# B&R Automation Studio project TD52 (part 99)

### module_GC.typ
```iecst
TYPE
	MM2VIS_Struct : 	STRUCT
		tCtrGenPF_Out : _tGeACtrOut; (* Controller to visulization out structure *) (*OldName:new pv;Cycle:5*)
		tCtr_Q_Out : _tGeACtrOut; (* Controller to visulization out structure *) (*OldName:new pv;Cycle:5*)
		bP_CosPCtr_Red_F_Hi : BOOL; (* power reduction by generator frequency high active *) (*OldName:bPowRedGenFrqH;Cycle:5*)
		bP_CosPCtr_Red_F_Lo : BOOL; (* power reduction by generator frequency low active *) (*OldName:bPowRedGenFrqL;Cycle:5*)
		bP_CosPCtr_Red_U_Hi : BOOL; (* power reduction by generator voltage high active *) (*OldName:bPowRedGenSpgH;Cycle:5*)
		bP_CosPCtr_Red_U_Lo : BOOL; (* power reduction by generator voltage low active *) (*OldName:bPowRedGenSpgL;Cycle:5*)
		bPF_Ctrl_Ena : BOOL; (* plant controller No. 13 enabled *) (*OldName:bPlantCtr13;Cycle:5*)
		rAng_CosPCtr_LimCalc : REAL; (* calculated limit polar wheel angle for power factor controller *) (*OldName:rQgLimit;Cycle:5*)
		rAng_CosPCtr_LimCalcVis : REAL; (*  Q- limit for visualization  *) (*OldName:ssQLimVis;Cycle:5*)
		rAng_CosPCtr_MinCalc : REAL; (* calculated minimum polar wheel angle for trip (LOSS OF EXCITATION) *) (*OldName:rQgErregerausfall;Cycle:5*)
		rAng_CosPCtr_MinCalcVis : REAL; (*  Q- trip limit for visualization  *) (*OldName:ssQTripVis;Cycle:5*)
		rP_Red_CosPCtr_F : REAL; (* power reduction by generator frequency *) (*OldName:ssPowerRedGenFrq;Cycle:5*)
		rP_Red_CosPCtr_T : REAL; (* power reduction by generator winding temperature *) (*OldName:ssPowerRedGenTemp;Cycle:5*)
		rP_Red_CosPCtr_U : REAL; (* power reduction by generator voltage *) (*OldName:ssPowerRedGenSpg;Cycle:5*)
		rP_Gen_ppt : REAL; (* nominal power in parts per thousand *) (*OldName:PN_PROM;Cycle:5*)
		rPF_CosPCtr_LimCalc1 : REAL; (* calculated reactive power trip limit of power 0 (zero) *) (*OldName:rQgTrip0;Cycle:5*)
		rPF_CosPCtr_LimCalc2 : REAL; (* calculated reactive power trip limit of nominal power 0 (PN_GASART) *) (*OldName:rQgTripN;Cycle:5*)
		rPF_CosPCtr_MinCalc1 : REAL; (* calculated reactive power limit of power 0 (zero) *) (*OldName:rQgLimit0;Cycle:5*)
		rPF_CosPCtr_MinCalc2 : REAL; (* calculated reactive power limit of nominal power 0 (PN_GASART) *) (*OldName:rQgLimitN;Cycle:5*)
		rPF_CosPCtr_Set_Ctr13 : REAL; (* set point value for plant controller *) (*OldName:ssContr_PF_SOLL;Cycle:5*)
		rPF_CosPCtr_Set_Vis : REAL; (* enable power factor input in visualization (picture 88) *) (*OldName:usPF_input_vis;Cycle:5*)
		rPF_CosPCtr_VisLine1 : REAL; (* value for visualization *) (*OldName:ucVisLine1_P14;Cycle:5*)
		rPF_GenCtr_Act : REAL; (* power factor generator controller actual value  *) (*OldName:ssContr_IST;Cycle:5*)
		rPF_GenCtr_Set : REAL; (* power factor generator controller set point  *) (*OldName:ssContr_SOLL;Cycle:5*)
		rQ_CosPCtr_Set : REAL; (* set point of reactive power for PF- controller on XT *) (*OldName:ssQSoll;Cycle:5*)
		rT_Gen_Bear_A_Act : REAL; (*Temperature generator bearing A*) (*OldName:ANA.LAG1;Cycle:5*)
		rT_Gen_Bear_B_Act : REAL; (*Temperature generator bearing B*) (*OldName:ANA.LAG2;Cycle:5*)
		rT_Gen_Wind_Act_L1 : REAL; (* generator winding temperature signal, winding phase 1 *) (*OldName:ANA.WICK1;Cycle:5*)
		rT_Gen_Wind_Act_L2 : REAL; (* generator winding temperature signal, winding phase 2 *) (*OldName:ANA.WICK2;Cycle:5*)
		rT_Gen_Wind_Act : REAL; (*generator winding temperature signal*) (*OldName:ANA.WICK;Cycle:;*)
		rU_Gen_Exc : REAL; (*Generator excitation voltage*) (*OldName:ANA.ERREG;Cycle:5;*)
		rT_Gen_Wind_Act_L3 : REAL; (* generator winding temperature signal, winding phase 3 *) (*OldName:ANA.WICK3;Cycle:5*)
		bOilSkid_Fan_Dem : BOOL; (*OilSkid - demand of fan (TRUE = on)*) (*OldName:newPv; Cycle:5;*)
		bOilSkid_Heater_Dem : BOOL; (*OilSkid - demand of heater (TRUE = on)*) (*OldName:newPv; Cycle:5;*)
		bOilSkid_PumpC_Dem : BOOL; (*OilSkid - demand of circulation pump (TRUE = on)*) (*OldName:newPv; Cycle:5;*)
		bOilSkid_PumpLP_Dem : BOOL; (*OilSkid - demand of low pressure pump (TRUE = on)*) (*OldName:newPv; Cycle:5;*)
		bOilSkid_PumpHP_Dem : BOOL; (*OilSkid - demand of high pressure pump (TRUE = on)*) (*OldName:newPv; Cycle:5;*)
		rPr_OilSkid_HP_DE : REAL; (*OilSkid - oil pressure in high pressure circuit to DE bearing [bar]*) (*OldName:newPv; Cycle:5;*)
		rPr_OilSkid_HP_NDE : REAL; (*OilSkid - oil pressure in high pressure circuit to NDE bearing [bar]*) (*OldName:newPv; Cycle:5;*)
		rT_OilSkid_Tank : REAL; (*OilSkid - tank temperature [°C]*) (*OldName:newPv; Cycle:5;*)
		rT_OilSkid_Supply : REAL; (*OilSkid - supply temperature [°C]*) (*OldName:newPv; Cycle:5;*)
		rLev_OilSkid_Tank : REAL; (*OilSkid - tank level [%]*) (*OldName:newPv; Cycle:5;*)
		rFlow_OilSkid_DE : REAL; (*OilSkid - oil flow to DE bearing [l/min]*) (*OldName:newPv; Cycle:5;*)
		rFlow_OilSkid_NDE : REAL; (*OilSkid - oil flow to NDE bearing [l/min]*) (*OldName:newPv; Cycle:5;*)
		rF_GenBear_DE1 : REAL; (*AI vibration generator bearing drive end 1*) (*Oldname:newPv;Cycle:5;*)
		rF_GenBear_DE2 : REAL; (*AI vibration generator bearing drive end 2*) (*Oldname:newPv;Cycle:5;*)
		rF_GenBear_NDE1 : REAL; (*AI vibration generator bearing non drive end 1*) (*Oldname:newPv;Cycle:5;*)
		rF_GenBear_NDE2 : REAL; (*AI vibration generator bearing non drive end 2*) (*Oldname:newPv;Cycle:5;*)
		rGen_T_In : REAL; (*AI generator air inlet temperature*) (*Oldname:t_GenAirIn;Cycle:5;*)
		rGen_T_In2 : REAL; (*AI generator air inlet temperature 2*) (*Oldname:newPv;Cycle:5;*)
		rT_GenAirOut : REAL; (*AI generator air outlet temperature*) (*Oldname:t_GenAirOut;Cycle:5;*)
		rQ_AVR_Set_Norm : REAL; (*reactive power setpoint [%]*) (*Oldname:newPv;Cycle:5;*)
		bSel_AVR_Set : BOOL; (*Q controller enabled*) (*Oldname:newPv;Cycle:5;*)
		bQ_Lim_On : BOOL; (*Q_Set is limited, Q_Limiter is working*) (*Oldname:newPv;Cycle:5;*)
		rQS_POC : REAL; (*Q/Sn diagram Y(graph)-value for point of control(POC)*) (*Oldname:newPv;Cycle:5;*)
		rPF_POC_Act_lin : REAL; (*PF diagram Y(graph)-value for point of control(POC)*) (*Oldname:newPv;Cycle:5;*)
		bU_Gen_Inc : BOOL; (* DI voltage adjustment external (increasing)*)
		bU_Gen_Dec : BOOL; (* DI voltage adjustment external (decreasing)*)
		bMsg1036 : BOOL; (*Generator over load/short circuit, Trip *) (*OldName:M_ULKS;Cycle:5*)
		bMsg1037 : BOOL; (*Generator winding temperature maximum, Trip *) (*OldName:AN_GWTA;Cycle:5*)
		bMsg1038 : BOOL; (*Generator reverse power, Trip *) (*OldName:M_RLSG;Cycle:5*)
		bMsg1062 : BOOL; (*measuring signal failure excitation voltage *) (*OldName:MS_EREG;Cycle:5*)
		bMsg1073 : BOOL; (*MMD: overload/short circuit *) (*OldName:ALM[1073];Cycle:5*)
		bMsg1109 : BOOL; (*loss of excitation (trip) *) (*OldName:bErregerAusfall;Cycle:5*)
		bMsg1110 : BOOL; (*Generator frequency low, Trip *) (*OldName:M_GFZN;Cycle:5*)
		bMsg1111 : BOOL; (*Generator frequency high, Trip *) (*OldName:M_GFZH;Cycle:5*)
		bMsg1112 : BOOL; (*Neutral current high, Trip *) (*OldName:M_INULL;Cycle:5*)
		bMsg1113 : BOOL; (*Generator power measuring signal failure*) (*OldName:M_PIST;Cycle:5*)
		bMsg1121 : BOOL; (* generator winding temperature maximum phase 1, Trip *) (*OldName:AN_GWA1;Cycle:5*)
		bMsg1122 : BOOL; (* generator winding temperature maximum phase 2, Trip *) (*OldName:AN_GWA2;Cycle:5*)
		bMsg1123 : BOOL; (* generator winding temperature maximum phase 3, Trip *) (*OldName:AN_GWA3;Cycle:5*)
		bMsg1124 : BOOL; (* generator bearing temperature maximum bearing A, Trip *) (*OldName:AN_LAGA1;Cycle:5*)
		bMsg1125 : BOOL; (* generator bearing temperature maximum bearing B, Trip *) (*OldName:AN_LAGA2;Cycle:5*)
		bMsg1126 : BOOL; (* generator voltage low, Trip *) (*OldName:M_GUZN;Cycle:5*)
		bMsg1127 : BOOL; (* generator voltage high, Trip *) (*OldName:M_GUZH;Cycle:5*)
		bMsg1132 : BOOL; (*Differential protection, Trip*) (*OldName:M_Diff;Cycle:5*)
		bMsg1134 : BOOL; (* Earth failure, Trip *) (*OldName:M_ERDS;Cycle:5*)
		bMsg1143 : BOOL; (* Voltage negative sequence (Voltage asymmetry), Trip *) (*OldName:M_UASY;Cycle:5*)
		bMsg1144 : BOOL; (* Current negative sequnece (Current asymmetrt), Trip *) (*OldName:M_IASY;Cycle:5*)
		bMsg1154 : BOOL; (* generator winding temperature maximum phase 1, Warning *) (*OldName:AN_GWW1;Cycle:5*)
		bMsg1155 : BOOL; (* generator winding temperature maximum phase 2, Warning *) (*OldName:AN_GWW2;Cycle:5*)
		bMsg1156 : BOOL; (* generator winding temperature maximum phase 3, Warning *) (*OldName:AN_GWW3;Cycle:5*)
		bMsg1157 : BOOL; (* generator bearing temperature maximum bearing A, Warning *) (*OldName:AN_LAGW1;Cycle:5*)
		bMsg1158 : BOOL; (* generator bearing temperature maximum bearing B, Warning *) (*OldName:AN_LAGW2;Cycle:5*)
		bMsg1185 : BOOL; (* generator winding temperature maximum, Warning *) (*OldName:AN_GWTW;Cycle:5*)
		bMsg2100 : BOOL; (* Differential protection, Warning *) (*OldName:M_STDIFF;Cycle:5*)
		bMsg2105 : BOOL; (* measuring signal failure winding temperature *) (*OldName:MS_GWT;Cycle:5*)
		bMsg2106 : BOOL; (* measuring signal failure winding temperature phase 1 *) (*OldName:MS_GWT1;Cycle:5*)
		bMsg2107 : BOOL; (* measuring signal failure winding temperature phase 2 *) (*OldName:MS_GWT2;Cycle:5*)
		bMsg2108 : BOOL; (* measuring signal failure winding temperature phase 3 *) (*OldName:MS_GWT3;Cycle:5*)
		bMsg2109 : BOOL; (* measuring signal failure bearing temperature bearing A *) (*OldName:MS_LAG1;Cycle:5*)
		bMsg2110 : BOOL; (* measuring signal failure bearing temperature bearing B *) (*OldName:MS_LAG2;Cycle:5*)
		bMsg2115 : BOOL; (* Generator voltage regulator failure *) (*OldName:Not-found;Cycle:5*)
		bMsg2156 : BOOL; (* B2156 Q-RED by winding temperature limit *) (*OldName:RPSDIA[35];Cycle:5*)
		bMsg2157 : BOOL; (* B2157 Q-limit by polar wheel angle *) (*OldName:RPSDIA[36];Cycle:5*)
		bMsg2202 : BOOL; (*generator DE bearing displacement*) (*OldName:newPv;Cycle:5*)
		bMsg2203 : BOOL; (*generator NDE bearing displacement*) (*OldName:newPv;Cycle:5*)
		bMsg2204 : BOOL; (*measuring signal failure displacement sensor 1 generator DE bearing*) (*OldName:newPv;Cycle:5*)
		bMsg2205 : BOOL; (*measuring signal failure displacement sensor 2 generator DE bearing*) (*OldName:newPv;Cycle:5*)
		bMsg2206 : BOOL; (*measuring signal failure displacement sensor 1 generator NDE bearing*) (*OldName:newPv;Cycle:5*)
		bMsg2207 : BOOL; (*measuring signal failure displacement sensor 2 generator NDE bearing*) (*OldName:newPv;Cycle:5*)
		bMsg2208 : BOOL; (*A2208 Oilskid tank oil level low *) (*OldName:newPv; Cycle:5;*)
		bMsg2209 : BOOL; (*not used - Generator Lube Oil System oil outlet pressure low*) (*OldName:newPv; Cycle:5;*)
		bMsg2210 : BOOL; (*not used - Generator both Lube Oil System AC oil pumps failed*) (*OldName:newPv; Cycle:5;*)
		bMsg2211 : BOOL; (*not used - Generator Lube Oil System oil supply temperature high*) (*OldName:newPv; Cycle:5;*)
		bMsg2212 : BOOL; (*not used - Generator both Jack Oil System AC oil pumps failed*) (*OldName:newPv; Cycle:5;*)
		bMsg2213 : BOOL; (*not used - Turbo charger oil filter differential pressure high*) (*OldName:newPv; Cycle:5;*)
		bMsg2235 : BOOL; (*not used - Generator Lube Oil System/Jack Oil System not ready*) (*OldName:newPv; Cycle:5;*)
		bMsg2277 : BOOL; (*Generator voltage too low 2*) (*OldName:newpv;Cycle:5*)
		bMsg2316 : BOOL; (*generator voltage high 2 (one phase)*) (*OldName:newPv;Cycle:5*)
		bMsg2336 : BOOL; (*Generator lube oil cooling system failure*) (*OldName:newpv;Cycle:5*)
		bMsg2371 : BOOL; (*A2371 Oil skid Oil flow to DE bearing Low*)
		bMsg2372 : BOOL; (*A2372 Oil skid Oil flow to NDE bearing Low*)
		bMsg2501 : BOOL; (*Generator rotating diode failure, Warning*) (*OldName:Not-found;Cycle:5*)
		bMsg2502 : BOOL; (*generator DE bearing displacement*) (*OldName:newPv;Cycle:5*)
		bMsg2503 : BOOL; (*generator NDE bearing displacement*) (*OldName:newPv;Cycle:5*)
		bMsg2504 : BOOL; (*Generator AVR panel MCB trip*) (*OldName:ALM[2504];Cycle:5*)
		bMsg2505 : BOOL; (*W2505 Oilskid low pressure oil filter clogged*) (*OldName:newPv; Cycle:5;*)
		bMsg2506 : BOOL; (*not used - Generator Lube Oil System pump A to B*) (*OldName:newPv; Cycle:5;*)
		bMsg2507 : BOOL; (*not used - Generator Lube Oil System pump B to A*) (*OldName:newPv; Cycle:5;*)
		bMsg2508 : BOOL; (*W2508 Oilskid high pressure oil filter DE clogged*) (*OldName:newPv; Cycle:5;*)
		bMsg2555 : BOOL; (*generator air inlet temperature*) (*OldName:newPv;Cycle:5*)
		bMsg2556 : BOOL; (*generator air outlet temperature*) (*OldName:newPv;Cycle:5*)
		bMsg2573 : BOOL; (* Overvoltage protection generator failure *) (*OldName:Not-found;Cycle:5*)
		bMsg2631 : BOOL; (*measuring signal failure displacement sensor 1 generator DE bearing*) (*OldName:newPv;Cycle:5*)
		bMsg2632 : BOOL; (*measuring signal failure displacement sensor 2 generator DE bearing*) (*OldName:newPv;Cycle:5*)
		bMsg2633 : BOOL; (*measuring signal failure displacement sensor 1 generator NDE bearing*) (*OldName:newPv;Cycle:5*)
		bMsg2634 : BOOL; (*measuring signal failure displacement sensor 2 generator NDE bearing*) (*OldName:newPv;Cycle:5*)
		bMsg2637 : BOOL; (*Generator interface panel circuit breaker tripped*) (*OldName:newPv;Cycle:5*)
		bMsg2665 : BOOL; (*Generator heater circuit breaker tripped*) (*OldName:newPv;Cycle:5*)
		bMsg2690 : BOOL; (*rotor earth fault*) (*OldName:newPV; Cycle:5;*)
		bMsg2691 : BOOL; (*reactive power/undervoltage protection (Q-U-protection)*) (*OldName:newPV; Cycle:5;*)
		bMsg2827 : BOOL; (*Generator Lube Oil System/Jacket Oil System read for start and operation*) (*OldName:bAMM[2827];Cycle:5;*)
		bMsg2828 : BOOL; (*Generator Lube Oil System oil outlet pressure ok*) (*OldName:bAMM[2828];Cycle:5;*)
		bMsg2829 : BOOL; (*Generator Lube Oil System drive end bearing oil flow ok*) (*OldName:bAMM[2829];Cycle:5;*)
		bMsg2830 : BOOL; (*Generator Lube Oil System non drive end bearing oil flow ok*) (*OldName:bAMM[2830];Cycle:5;*)
		bMsg2998 : BOOL; (*Q-limit by under voltage*)
		bMsg3219 : BOOL; (* excitation voltage low *) (*OldName:AN_ERGW1;Cycle:5*)
		bMsg3298 : BOOL; (* gcb opened by generator reverse power  *) (*OldName:ALM[3298];Cycle:5*)
		bMsg3299 : BOOL; (* gcb opened by current negative sequence *) (*OldName:ALM[3299];Cycle:5*)
		bMsg3319 : BOOL; (* generator protection trip *) (*OldName:ALM[3319];Cycle:5*)
		bMsg3393 : BOOL; (*generator overexcitation*) (*OldName:newPV; Cycle:5;*)
		bMsg3418 : BOOL; (*W3418 Oilskid oil in oil sump *) (*OldName:newPv; Cycle:5;*)
		bMsg3419 : BOOL; (*W3419 Oilskid tank oil level measuring signal failure *) (*OldName:newPv; Cycle:5;*)
		bMsg3420 : BOOL; (*W3420 Oilskid tank oil level low*) (*OldName:newPv; Cycle:5;*)
		bMsg3421 : BOOL; (*W3421 Oilskid tank oil temperature measuring signal failure*) (*OldName:newPv; Cycle:5;*)
		bMsg3422 : BOOL; (*W3422 Oilskid tank oil temperature low*) (*OldName:newPv; Cycle:5;*)
		bMsg3423 : BOOL; (*W3423 Oilskid oil supply temperature measuring signal failure*) (*OldName:newPv; Cycle:5;*)
		bMsg3424 : BOOL; (*W3424 Oilskid oil supply temperature low*) (*OldName:newPv; Cycle:5;*)
		bMsg3425 : BOOL; (*W3425 Oilskid oil supply temperature high*) (*OldName:newPv; Cycle:5;*)
		bMsg3426 : BOOL; (*W3426 Oilskid low pressure oil pump circuit breaker tripped*) (*OldName:newPv; Cycle:5;*)
		bMsg3427 : BOOL; (*W3427 Oilskid oil flow TO DE bearing measuring signal failure*) (*OldName:newPv; Cycle:5;*)
		bMsg3428 : BOOL; (*W3428 Oilskid oil flow TO DE bearing low*) (*OldName:newPv; Cycle:5;*)
		bMsg3429 : BOOL; (*W3429 Oilskid oil flow TO DE bearing high*) (*OldName:newPv; Cycle:5;*)
		bMsg3430 : BOOL; (*W3430 Oilskid oil flow TO NDE bearing measuring signal failure*) (*OldName:newPv; Cycle:5;*)
		bMsg3431 : BOOL; (*W3431 Oilskid oil flow TO NDE bearing low*) (*OldName:newPv; Cycle:5;*)
		bMsg3432 : BOOL; (*W3432 Oilskid oil flow TO NDE bearing high*) (*OldName:newPv; Cycle:5;*)
		bMsg3433 : BOOL; (*W3433 Oilskid high pressure oil pump circuit breaker tripped*) (*OldName:newPv; Cycle:5;*)
		bMsg3434 : BOOL; (*W3434 Oilskid high pressure oil pump circuit breaker tripped - UPS*) (*OldName:newPv; Cycle:5;*)
		bMsg3435 : BOOL; (*W3435 Oilskid oil pressure TO DE bearing measuring signal failure*) (*OldName:newPv; Cycle:5;*)
		bMsg3436 : BOOL; (*W3436 Oilskid oil pressure TO DE bearing low*) (*OldName:newPv; Cycle:5;*)
		bMsg3442 : BOOL; (*W3442 Oilskid oil pressure TO NDE bearing measuring signal failure*) (*OldName:newPv; Cycle:5;*)
		bMsg3443 : BOOL; (*W3443 Oilskid oil pressure TO NDE bearing low*) (*OldName:newPv; Cycle:5;*)
		bMsg3446 : BOOL; (*W3446 Oilskid high pressure oil filter NDE clogged*) (*OldName:newPv; Cycle:5;*)
		bMsg3437 : BOOL; (*W3437 Oilskid fan circuit breaker tripped*) (*OldName:newPv; Cycle:5;*)
		bMsg3438 : BOOL; (*W3438 Oilskid heater circuit breaker tripped*) (*OldName:newPv; Cycle:5;*)
		bMsg3439 : BOOL; (*W3439 Oilskid main switch auxiliaries opened*) (*OldName:newPv; Cycle:5;*)
		bMsg3440 : BOOL; (*W3440 Oilskid auxiliaries voltage NOT available*) (*OldName:newPv; Cycle:5;*)
		bMsg3441 : BOOL; (*W3441 Oilskid auxiliaries voltage NOT available - UPS*) (*OldName:newPv; Cycle:5;*)
		bMsg3447 : BOOL; (*W3447 Oilskid circulation pump circuit breaker tripped*) (*OldName:newPv; Cycle:5;*)
		bMsg3468 : BOOL; (*generator air inlet temperature 2 signal failure*) (*OldName:newPv;Cycle:5*)
		bMsg3516 : BOOL; (*excitation voltage high*) (*OldName:AN_ERGW2;Cycle:5*)
		bMsg3563 : BOOL; (*Generator lubrication failure, Warning*) (*OldName:Not-found;Cycle:5*)
		bMsg3566 : BOOL; (*Generator power factor setpoint measuring signal failur*) (*Oldname: ALM[3566];Cycle:5*)
		bMsg3573 : BOOL; (*Generatow lube oil cooling system failure*) (*OldName:newpv;Cycle:5*)
		bMsg9311 : BOOL; (*Earth failure, warning*)
		tU_Stat : _tXY_Stat; (* Voltage static XY Diagram *)
		bCntGndFail_Visible : BOOL; (*counter earth failure visibility*)
		bMsg1038Set : BOOL; (*Generator reverse power, Trip*)
		bMsg1109Set : BOOL; (*loss of excitation (trip)*)
		bMsg1110Set : BOOL; (*Generator frequency low, Trip*)
		bMsg1111Set : BOOL; (*Generator frequency high, Trip*)
		bMsg1112Set : BOOL; (*Neutral current high, Trip*)
		bMsg1126Set : BOOL; (*generator voltage low, Trip*)
		bMsg1127Set : BOOL; (*generator voltage high, Trip*)
		bMsg1143Set : BOOL; (*Voltage negative sequence (Voltage asymmetry), Trip*)
		bMsg1144Set : BOOL; (*Current negative sequnece (Current asymmetrt), Trip*)
		bMsg2277Set : BOOL; (*Generator voltage too low 2*)
		bMsg2316Set : BOOL; (*generator voltage high 2 (one phase)*)
		bMsg9351 : BOOL; (*Measuring signal failure external reactive power set point for voltage droop mode*)
		bMsg9365 : BOOL; (*Automatic generator greasing system error (drive end DE bearing) *)
		bMsg9366 : BOOL; (*Automatic generator greasing system error (non-drive end NDE bearing) *)
		bMsg9367 : BOOL; (*Automatic generator greasing system - lubrication cartridge empty (drive end DE bearing) *)
		bMsg9368 : BOOL; (*Automatic generator greasing system - lubrication cartridge empty (non-drive end NDE bearing) *)
		rQ_Droop_Offs : REAL; (*Actual reactive power set point for voltage droop mode*)
		iIdx_Q_Droop_Offs : INT; (*Source of reactive power set point for voltage droop mode 0=none/1=analog/2=bus/3=HMI)*)
		iSource_U_OffsSet : INT; (* Voltage setpoint in island mode: 0= no setpoint, 1= Droop, 2= External *)
		bMsg9372 : BOOL; (*W9372 Multi measurement device: Earth failure generator*)
		bMsg2373 : BOOL; (*A2373 Multi measurement device: Earth failure generator*)
	END_STRUCT;
END_TYPE

(*END_MM2VIS*)

TYPE
	VIS2MM_Struct : 	STRUCT
		tCtrGenPF_In : _tGeACtrIn; (*Visulization to Controller in structure*) (*OldName:new pv;Cycle:5*)
		tCtr_Q_In : _tGeACtrIn; (*Visulization to Controller in structure*) (*OldName:new pv;Cycle:5*)
		iCnt_OilSkid_HP_PrErr : INT; (*Para-Visu synchronization operating mode selection*) (*OldName:newPv; Cycle:5;*)
		iOpH_GndFailure : DINT; (* earth failure h *)
		bQ_Droop_Set_Man : BOOL; (*Manual reactive power set point for voltage droop mode active*)
		rQ_Droop_Set_Man : REAL; (*Manual reactive power set point for voltage droop mode active*)
	END_STRUCT;
	IN_GC_Struct : 	STRUCT
		tAB2GC : AmmBase2MM; (*Structure Alarm base to Generator control module*) (*OldName:new pv;Cycle:5;*)
		tPB2MM : ParaBase2MM_type; (*Data exchange structure to ParaBase*) (*OldName:new PV;Cycle:5*)
		tCustAnaIn : ARRAY[0..120]OF HALioAi_Type; (*Replacement for RAN_KANAL...*) (*OldName: ANA_RAN; Cycle:5;*)
		tCustDigIn : ARRAY[0..200]OF HALioDi_Type; (*new, reserved for Project specific use*) (*OldName: newPV; Cycle:5;*)
		tExtCtrOk : HALioDi_Type; (* DI: External speed / voltage controller okay *) (*OldName: newPV; Cycle:5;*)
		tECWP_PreH_Dem : HALioDo_Type; (*engine cooling water preheating pump demand*) (*OldName:A_VORW;Cycle:5*)
		tEleStarter_Dem : HALioDo_Type; (*electric starter demand*) (*OldName:A_STRT;Cycle:5;*)
		tU_Gen_Dec : HALioDi_Type; (*digital input for voltage adjustment external (decreasing)*) (*OldName:DI_u_minus; Cycle: 5;*)
		tU_Gen_Inc : HALioDi_Type; (*digital input for voltage adjustment external (increasing)*) (*OldName:DI_u_plus; Cycle: 5;*)
		tDiffPrct : HALioDi_Type; (*DI: Differential protection *) (*OldName:DIFF;Cycle:5*)
		tEng_Run : HALioDo_Type; (*Engine in operation*) (*OldName:M_BTRB;Cycle:5*)
		tEng_SUExc_Rel : HALioDi_Type; (*start-up excitation release*) (*OldName:U_SY_LFG;Cycle:5*)
		tF_MMD : ARRAY[0..2]OF HALioAi_Type; (*actual generator frequency*) (*OldName:usFreq,ssFreq;Cycle:5*)
		tF_MMD_LimHi : ARRAY[0..2]OF HALioDi_Type; (*generator frequency too high*) (*OldName:GFZH;Cycle:5*)
		tF_MMD_LimLo : ARRAY[0..2]OF HALioDi_Type; (*generator frequency too low*) (*OldName:GFZN;Cycle:5*)
		tFlow_Gen_Lube : HALioDi_Type; (*generator lubrication failure*) (*OldName:DI_GENS_F ;Cycle:5*)
		tGCB_DVM : HALioDi_Type; (*voltage matching for synchronization*) (*OldName:MSY_DVM;Cycle:5*)
		tGCB_On : HALioDi_Type; (*Generator circuit breaker*) (*OldName:GCB_ON;Cycle:5*)
		tGen_Exc_Off : HALioDi_Type; (*de- excitation*) (*OldName:T_ENTR;Cycle:5*)
		tGen_T_In : HALioAi_Type; (*generator air inlet temperature*) (*OldName:t_GenAirIn;Cycle:5*)
		tGen_T_In2 : HALioAi_Type; (*generator air inlet temperature*) (*OldName:new_pv;Cycle:5*)
		tT_GenAirOut : HALioAi_Type; (*generator air outlet temperature*) (*OldName:t_GenAirOut;Cycle:5*)
		tGenDeexitDem : HALioDo_Type; (*generator deexitation demand*) (*OldName:A_ENTR;Cycle:5*)
		tGenPrctTrip : HALioDi_Type; (*Generator protection trip*) (*OldName:DI_GEN_PT_TC1;Cycle:5*)
		tGndFailure : HALioDi_Type; (*earth failure generator*) (*OldName:ERDS;Cycle:5*)
		tI_Diff : HALioDi_Type; (*generator differential protection trip*) (*OldName:ST_DIFF;Cycle:5*)
		tI_MMD_Asy : ARRAY[0..2]OF HALioDi_Type; (*generator current negative sequence too high*) (*OldName:IASY;Cycle:5*)
		tI_MMD_LimHi : HALioDi_Type; (*MMD: overload short circuit*) (*OldName:DI_MMD_OL_TC1;Cycle:5*)
		tI_MMD_Neutr_LimHi : ARRAY[0..2]OF HALioDi_Type; (*generator neutral current too high*) (*OldName:INULL;Cycle:5*)
		tMCB_On : HALioDi_Type; (*mains circuit breaker closed*) (*OldName:MCB_ON;Cycle:5*)
		tOlShortCirc : HALioDi_Type; (*Overload/short circuit*) (*OldName:ULKS, DI_GCB_OL_TC1;Cycle:5*)
		tP_Act : ARRAY[0..2]OF HALioAi_Type; (*actual electric power [kW] *) (*OldName:ssPAct;Cycle:5*)
		tPF_Act : ARRAY[0..2]OF HALioAi_Type; (*actual cos phi value *) (*OldName:ssCosPhi, ANA.COSPHI;Cycle:5*)
		tQ_Act : ARRAY[0..2]OF HALioAi_Type; (*actual reactive power [kVar] *) (*OldName:ssPReac;Cycle:5*)
		tRel_U_Sel_LS_Gen : HALioDi_Type; (*Release voltage selection LS-Generator *) (*OldName:E_LSHK;Cycle:5*)
		tReq_PowMod : HALioDi_Type; (*request power operation mode *) (*OldName:DI_DMND_PM;Cycle:5*)
		tT_Gen_Bear_A_Act : HALioAi_Type; (*generator bearing A temperature signal*) (*OldName:ANA.LAG1;Cycle:5*)
		tT_Gen_Bear_B_Act : HALioAi_Type; (*generator bearing B temperature signal*) (*OldName:ANA.LAG2;Cycle:5*)
		tT_Gen_Wind : HALioAi_Type; (*actual generator winding temperature signal*) (*OldName:ANA.WICK;Cycle:5*)
		tT_Gen_Wind_Act_L1 : HALioAi_Type; (*generator winding temperature signal, winding phase 1*) (*OldName:ANA.WICK1;Cycle:5*)
		tT_Gen_Wind_Act_L2 : HALioAi_Type; (*generator winding temperature signal, winding phase 2*) (*OldName:ANA.WICK2;Cycle:5*)
		tT_Gen_Wind_Act_L3 : HALioAi_Type; (*generator winding temperature signal, winding phase 3*) (*OldName:ANA.WICK3;Cycle:5*)
		tU_Adj_Minus : HALioDi_Type; (*Voltage adjustment Minus *) (*OldName:A_UMIN;Cycle:5*)
		tU_Adj_Plus : HALioDi_Type; (*Voltage adjustment Plus *) (*OldName:A_UPLU;Cycle:5*)
		tU_Avg : ARRAY[0..2]OF HALioAi_Type; (*actual generator average voltage*) (*OldName:ssUAvg;Cycle:5*)
		tU_Gen_Contr_Fail : HALioDi_Type; (*generator voltage regulator failure *) (*OldName:DI_GENREG_F;Cycle:5*)
		tU_Gen_Exc : HALioAi_Type; (*actual excitation voltage signal, filtered and scaled*) (*OldName:ANA.ERREG;Cycle:5*)
		tU_Gen_LimHi : ARRAY[0..2]OF HALioDi_Type; (*generator voltage too high*) (*OldName:GUZH ;Cycle:5*)
		tU_Gen_LimLo2 : ARRAY[0..2]OF HALioDi_Type; (*generator voltage too low 2*) (*OldName:GUZN_2;Cycle:5*)
		tU_Gen_LimLo : ARRAY[0..2]OF HALioDi_Type; (*generator voltage too low*) (*OldName:GUZN;Cycle:5*)
		tU_GenDiode_Fail : HALioDi_Type; (*generator diode alarm*) (*OldName:DI_GEN_D_F ;Cycle:5*)
		tU_GenDiode_Trip : HALioDi_Type; (*generator diode trip*) (*OldName:DI_GEN_D_Tr ;Cycle:5*)
		tU_GenOverVolt : HALioDi_Type; (*failure generator overvoltage protection*) (*OldName:DI_GOVP ;Cycle:5*)
		tGen_LO_CoolingSys_Fail : HALioDi_Type; (*generator lube oil cooling system failure*) (*OldName: DI_GEN_BERC; Cycle: 5;*)
		tGenCtr_CktBkr_Trip : HALioDi_Type; (*generator cicuit breaker off*) (*OldName: GEN_AVR_CB; Cycle: 5;*)
		tU_MMD_Asy : ARRAY[0..2]OF HALioDi_Type; (*generator voltage negative sequence too high*) (*OldName:UASY;Cycle:5*)
		tU_MMD_Synch1 : ARRAY[0..2]OF HALioAi_Type; (*phase voltage system 1*) (*OldName:ssSynch1Volt;Cycle:5*)
		tU_MMD_Synch2 : ARRAY[0..2]OF HALioAi_Type; (*phase voltage system 2*) (*OldName:ssSynch2Volt;Cycle:5*)
		rT_Ch_T1LP_Avg : REAL; (*average charge temperature before low-pressure turbocharger (= engine intake air) [°C]*) (*OldName:ssIATemp,ANA_ZLTP,tT_InAirER; Cycle:5;*) (* V04.04.00.00 *)
		bAMM_T_Ch_T1LP_Avg : BOOL; (*collective warning - average charge temp. before low-pressure TC (= engine intake air)*) (* V04.04.00.00 *)
		bECW_Gnl_PreH_Dem : BOOL; (*engine cooling water preheating demand *)
		tLev_OilSkid_Sump_Hi : HALioDi_Type; (*OilSkid oil in safety sump *) (*Oldname:new pv;Cycle:5;*)
		tOilSkid_PumpLP_CBOk : HALioDi_Type; (*OilSkid low pressure pump - circuit breaker*) (*Oldname:new pv;Cycle:5;*)
		tDPr_OilSkid_FiltLP_Hi : HALioDi_Type; (*OilSkid difference pressure - oil low pressure filter*) (*Oldname:new pv;Cycle:5;*)
		tOilSkid_PumpHP_DemOn : HALioDi_Type; (*OilSkid high pressure pump - demand ON*) (*Oldname:new pv;Cycle:5;*)
		tOilSkid_PumpHP_DemOff : HALioDi_Type; (*OilSkid high pressure pump - demand OFF*) (*Oldname:new pv;Cycle:5;*)
		tOilSkid_PumpHP_CBOk : HALioDi_Type; (*OilSkid high pressure pump - circuit breaker*) (*Oldname:new pv;Cycle:5;*)
		tOilSkid_PumpHP_CBOk_UPS : HALioDi_Type; (*OilSkid high pressure pump - circuit breaker UPS*) (*Oldname:new pv;Cycle:5;*)
		tT_OilSkid_Supply : HALioAi_Type; (*OilSkid supply temperature*) (*Oldname:new pv;Cycle:5;*)
		tT_OilSkid_Tank : HALioAi_Type; (*OilSkid tank temperature*) (*Oldname:new pv;Cycle:5;*)
		tLev_OilSkid_Tank : HALioAi_Type; (*OilSkid tank level*) (*Oldname:new pv;Cycle:5;*)
		tFlow_OilSkid_DE : HALioAi_Type; (*OilSkid oil flow to DE bearing *) (*Oldname:new pv;Cycle:5;*)
		tFlow_OilSkid_NDE : HALioAi_Type; (*OilSkid oil flow to NDE bearing (G.03-FI-003)*) (*Oldname:new pv;Cycle:5;*)
		tOilSkid_Heater_CBOk : HALioDi_Type; (*OilSkid heater - circuit breaker*) (*Oldname:new pv;Cycle:5;*)
		tDPr_OilSkid_FiltHP_DE_Hi : HALioDi_Type; (*OilSkid difference pressure - oil high pressure filter to DE bearing*) (*Oldname:new pv;Cycle:5;*)
		tDPr_OilSkid_FiltHP_NDE_Hi : HALioDi_Type; (*OilSkid difference pressure - oil high pressure filter to NDE bearing*) (*Oldname:new pv;Cycle:5;*)
		tOilSkid_Fan_CBOk : HALioDi_Type; (*OilSkid fan - circuit breaker*) (*Oldname:new pv;Cycle:5;*)
		tOilSkid_MCB : HALioDi_Type; (*OilSkid main switch auxiliaries opened*) (*Oldname:new pv;Cycle:5;*)
		tOilSkid_AuxV_Ok : HALioDi_Type; (*OilSkid auxiliaries voltage not available*) (*Oldname:new pv;Cycle:5;*)
		tOilSkid_AuxV_Ok_UPS : HALioDi_Type; (*OilSkid auxiliaries voltage not available - UPS*) (*Oldname:new pv;Cycle:5;*)
		tOilSkid_PumpC_CBOk : HALioDi_Type; (*OilSkid circulation pump - circuit breaker*) (*Oldname:new pv;Cycle:5;*)
		tPr_OilSkid_HP_DE : HALioAi_Type; (*OilSkid oil pressure in high pressure circuit to DE bearing*) (*Oldname:new pv;Cycle:5;*)
		tPr_OilSkid_HP_NDE : HALioAi_Type; (*OilSkid oil pressure in high pressure circuit to NDE bearing *) (*Oldname:new pv;Cycle:5;*)
		tF_GenBear_DE1 : HALioAi_Type; (*vibration generator bearing drive end 1*) (*Oldname:AI_v_GenBearDE1;Cycle:5;*)
		tF_GenBear_DE2 : HALioAi_Type; (*vibration generator bearing drive end 2*) (*Oldname:AI_v_GenBearDE2;Cycle:5;*)
		tF_GenBear_NDE1 : HALioAi_Type; (*vibration generator bearing non drive end 1*) (*Oldname:AI_v_GenBearNDE1;Cycle:5;*)
		tF_GenBear_NDE2 : HALioAi_Type; (*vibration generator bearing non drive end 2*) (*Oldname:AI_v_GenBearNDE2;Cycle:5;*)
		tGenIF_CB_On : HALioDi_Type; (*Generator interface panel circuit breaker tripped*) (*Oldname:DI_GENI_CB_trip;Cycle:5;*)
		tGenHeat_CB_On : HALioDi_Type; (*Generator heater circuit breaker tripped*) (*Oldname:newPv;Cycle:5;*)
		bEng_RPSDem : BOOL; (*engine demanded  *) (*OldName:A_AGFD; Cycle:5*)
		rCust_SparePara : ARRAY[0..200]OF REAL; (*SPS_REZP1 to SPS_REZP200	*) (* OldName: SPS_REZP1, SPS_REZP2, SPS_REZP70; Cycle: 5; *)
		iGCQ_Fun_Act : USINT; (*Number of the active Voltage control function from static GridCode*) (*OldName:usGCQ_Fun_act;Cycle:5*)
		bGCQ_Fun_Act : BOOL; (* falls eigenes Modul Schnittstelle zu reg_in(_9) - stat. GC Funktion aktiv *) (* OldName: bGCQ_Fun_act; Cycle: 0 *)
		rPFSoll_lin_GR2GC : REAL; (*power factor setpoint GR->GC incl.QLim + GR/EVU_funct.1-5*) (*OldName:newPV;Cycle:5*)
		bScavFinished : BOOL; (*scavenging cycle finished *) (*OldName:SPUEL_AB; Cycle:5;*)
		bEO_PrelubeDemIgn : BOOL; (*Demand Prelubricating from ignition*) (*OldName:PRELUBE_IgnST; Cycle:5;*)
		bEng_Aux_Dem : BOOL; (*engine auxiliaries demand *) (*OldName:M_ANFHBT;Cycle:5;*)
		bEng_Dem : BOOL; (*Module demanded*) (*OldName:M_AGFD;Cycle:5;*)
		bEng_Dem_EPS : BOOL; (*engine demand for emergency operation*) (*OldName:M_NANF;Cycle:5;*)
		bEng_Start : BOOL; (*Engine start command*) (*OldName:M_STRT;Cycle:5;*)
		bGCB_DemSy : BOOL; (*generator circuit breaker demand synchronization*) (*OldName:ASYANW;Cycle:5;*)
		bGen_SyD_Dem : BOOL; (* demand synch.device *) (*OldName:dmnd_sy_device;Cycle:5;*)
		bGV_On : BOOL; (*command open gas valves*) (*OldName:M_GASV;Cycle:5;*)
		bIgn_Dem : BOOL; (*Demand ignition*) (*OldName:ZUEND;Cycle:5;*)
		bMCB_DemSy : BOOL; (*mains circuit breaker demand synchronization*) (*OldName:ARSYANW;Cycle:5;*)
		bOtherGenParallel : BOOL; (*1 Genset still in operation and demanded *) (*OldName:PARALLEL;Cycle:5;*)
		bSCO_Active : BOOL; (*safety cut out gas valves glow ignition prevention*) (*OldName:SICH_SCHL;Cycle:5;*)
		bSynchDem : BOOL; (*synchronization demanded*) (*OldName:bSynch;Cycle:5;*)
		bSyncSlipMode : ARRAY[0..2]OF BOOL; (* MMD synchronization with slip mode *) (*OldName:bSyncSlipMode;Cycle:5;*)
		iIdx_Gtyp_Dem : INT; (* actual gassort 0 to 4 *) (*OldName:gasart;Cycle:5;*)
		iSt_OpMode : UDINT; (*Operating mode*) (*OldName:InselM;Cycle:5;*)
		iIdx_OMSS : INT; (*Index of operation mode selector switch*) (*OldName:BWS_HA ;Cycle:5;*)
		rN_EngAct : REAL; (* Engine Speed (1/min) *) (*OldName:ANA.DREHZ;Cycle:5;*)
		rP_Act_Norm_Filt : REAL; (*Actual normalized power*) (*OldName:P_IST_PROM;Cycle:5;*)
		rP_Act_Norm : REAL; (*actual power related to rP_Nom without filter *) (* OldName: P_IST_OF; Cyclic:5; *)
		rP_Nom : REAL; (*Nominal power*) (*OldName:PN_GASART;Cycle:5;*)
		rPF_CosPCtr_Bus : REAL; (*Power factor setpoint via bus*) (*Oldname:new pv;Cycle:5;*)
		bEng_Aux_Dem_CDR : BOOL; (*engine auxiliaries demand with cool down run*) (*OldName:ANFHBT; Cycle:5*)
		bMsg1031 : BOOL; (*Emergency stop*) (*OldName: M_SIS; Cycle: 5;*)
		bMsg1054 : BOOL; (*Fire alarm*) (*OldName:M_BAL; Cycle: 5;*)
		tP_GenRev_Ext : HALioDi_Type; (*generator reverse power*) (*OldName:newPV; Cycle:5*)
		tGenLossExc_Ext : HALioDi_Type; (*generator loss of excitation*) (*OldName:newPV; Cycle:5*)
		tU_GenAsy_Ext : HALioDi_Type; (*voltage negative sequence*) (*OldName:newPV; Cycle:5*)
		tI_GenAsy_Ext : HALioDi_Type; (*current negative sequence*) (*OldName:newPV; Cycle:5*)
		tGenOverExc : HALioDi_Type; (*generator overexcitation*) (*OldName:newPV; Cycle:5*)
		tGenRotorEarthFault : HALioDi_Type; (*rotor earth fault*) (*OldName:newPV; Cycle:5*)
		tQ_GenUnderVoltProt : HALioDi_Type; (*reactive power/undervoltage protection (Q-U-protection)*) (*OldName:newPV; Cycle:5*)
		bMMD_GenAlarmTestOn : BOOL; (*MMD_Gen alarm test On*) (*OldName:newPv; Cycle:5;*)
		bN2_ScavCoPrelubeOn : BOOL; (*N2 scavenging command prelubrication ON*) (*OldName:PRELUBE_SC;Cycle:5*)
		bTP_GrC_Event : BOOL;
		bOilskidDemSTFS : BOOL; (*oilskid demand for slowturn faststart*) (* Oldname: new PV, Cycle:5 *)
		tS_Act : ARRAY[0..2]OF HALioAi_Type; (*actual aparent power [kVar] *) (*OldName:newPV;Cycle:5*)
		rQSoll_filt_GR2GC : REAL; (*Q setpoint after ramp before limiter from GR*) (*OldName:newPV;Cycle:5*)
		rQSoll_Lim_GR2GC : REAL; (*Q setpoint limited from GR*) (*OldName:newPV;Cycle:5*)
		rP_POC_Act_Cust : REAL; (*active power actual  from customer(point of connection)[kW]*) (*OldName:newPV;Cycle:5*)
		rS_POC_Act_Cust : REAL; (*apparent power actual from customer(point of connection)[kVA]*) (*OldName:newPV;Cycle:5*)
		rQ_POC_Act_Cust : REAL; (*reactive power actual from customer(point of connection)[kVAr]*) (*OldName:newPV;Cycle:5*)
		rPF_POC_Act_Cust : REAL; (*power factor actual from customer(point of connection)*) (*OldName:newPV;Cycle:5*)
		bQSetLim : BOOL; (*GR: Q limitation custom OR Q(U) ON*) (*OldName:newPV;Cycle:5*)
		tU_L1L2 : ARRAY[0..2]OF HALioAi_Type; (* generator voltage phase 1_2 [V] *) (*OldName:ssUL1L2[1];Cycle:5;*)
		tU_L2L3 : ARRAY[0..2]OF HALioAi_Type; (* generator voltage phase 2_3 [V] *) (*OldName:ssUL2L3[1];Cycle:5;*)
		tU_L3L1 : ARRAY[0..2]OF HALioAi_Type; (* generator voltage phase 3_1 [V] *) (*OldName:ssUL3L1[1];Cycle:5;*)
		tU_L1N : ARRAY[0..2]OF HALioAi_Type; (* generator voltage phase 1_N [V] *) (*OldName:ssUL1N[1];Cycle:5;*)
		tU_L2N : ARRAY[0..2]OF HALioAi_Type; (* generator voltage phase 2_N [V] *) (*OldName:ssUL2N[1];Cycle:5;*)
		tU_L3N : ARRAY[0..2]OF HALioAi_Type; (* generator voltage phase 3_N [V] *) (*OldName:ssUL3N[1];Cycle:5;*)
		rU_Set_Norm_Cust : REAL; (* External voltage set point from CU module [%Unom] *) (*OldName:new PV V4.07;Cycle:5*)
		bMsg2831 : BOOL; (* B2831 Low Voltage Ride Through Event *)
		tGndFaultW : HALioDi_Type; (*Earth failure generator warning*)
		bN_U_Set_Ext_On : BOOL; (*External speed and voltage control ON*)
		tQ_Droop_Set : HALioAi_Type; (*reactive power setpoint in voltage droop*)
		tU_SetExtAI_Norm : HALioAi_Type; (*setpoint voltage [%Unom]*)
		rQset_Droop_Bus : REAL; (*Reactive power setpoint for droop mode via Bus*)
		rUset_Isl_Bus : REAL; (*Generator voltage setpoint via Bus*)
		bMsg1147 : BOOL; (*W1147 Outage coupling with central control system*)
		bExtCtrOk : BOOL; (*External voltage/speed control released*)
		rU_Set_NP : REAL; (*voltage setpoint-net parallel mode*)
		bU_Set_NP_Rel : BOOL; (*voltage setpoint-net parallel mode/release*)
		tGenBearGreasSys2DE : HALioDi_Type; (*INNIO STAR CONTROL SYSTEM Pin2 drive end DE bearing*)
		tGenBearGreasSys4DE : HALioDi_Type; (*INNIO STAR CONTROL SYSTEM Pin4 drive end DE bearing*)
		tGenBearGreasSys2NDE : HALioDi_Type; (*INNIO STAR CONTROL SYSTEM Pin2 non-drive end NDE bearing*)
		tGenBearGreasSys4NDE : HALioDi_Type; (*INNIO STAR CONTROL SYSTEM Pin4 non-drive end NDE bearing*)
		bGCB_aut_on2dead_bb : BOOL; (*generator circuit breaker automatic on to dead bus bar*)
		iTimeStamp_PosZeroCrossing_UGen1 : DINT; (*TimeStamp of last positive zero crossing UGen1 [ 1 / 4096microseconds]*)
		iTimeStamp_PosZeroCrossing_UGen2 : DINT; (*TimeStamp of last positive zero crossing UGen2 [ 1 / 4096microseconds]*)
		iTimeStamp_PosZeroCrossing_UGen3 : DINT; (*TimeStamp of last positive zero crossing UGen3 [ 1 / 4096microseconds]*)
		bReq_PowMod : BOOL; (*request power mode - over-written in customization*)
		bBypassMCB_CosPhi : BOOL; (*bypass MCB status information from the standard CosPhi Ctrl check*)
		bSimWinMOD_Active : BOOL; (*WinMode simulation active *) (*OldName:new PV; Cycle:5*)
	END_STRUCT;
END_TYPE

(*END_IN*)

TYPE
	OUT_GC_Struct : 	STRUCT
		tGC2AB : MM2AmmBase; (*AMM structure *) (*OldName:new pv;Cycle:5*)
		tGC2PB : MM2ParaBase_type; (*Data exchange structure to ParaBase*) (*OldName:new pv;Cycle:5*)
		tPF_AO_PF_U : HALioAo_Type; (*power factor generator *) (* OldName:AO_PF_gen_V;Cycle:5*)
		tPF_AO_PF_I : HALioAo_Type; (*power factor generator *) (* OldName:AO_PF_gen_mA;Cycle:5*)
		tGen_PreHDem : HALioDo_Type; (*Generator preheat demand*) (*OldName: DO_GenPreH; Cycle:5;*)
		tCtr_Gen_Set : HALioAo_Type; (*Generator ???*) (*OldName:new pv;Cycle:5*)
		tGCB_On_ReturnSign : HALioDo_Type; (*Release for Unitrol AVR*) (*Oldname:DO_GCB_ON;Cycle:5*)
		tLOS_Dem : HALioDo_Type; (*Generator demand lube oil system*) (*OldName:DO_GEN_BERC;Cycle:5*)
		tLeroySomer_AuxContactor : HALioDo_Type; (*LEROY-SOMER Auxiliary Contactor *) (*OldName:LSHK;Cycle:5*)
		tPF_CosPCtr_Ena : HALioDo_Type; (*power factor controller enabled*) (*OldName:A_COSPHI;Cycle:5*)
		tT_AO_Gen_T_In : HALioAo_Type; (*Generator air inlet temperature for gen.controler*) (*OldName:AO_t_GenAirIn_V;Cycle:5*)
		tGenCtrResetSp : HALioDo_Type; (*Generator controller reset setpoint*) (*OldName:DO_GenCtrResetSp;Cycle:5*)
		tU_MidPos : HALioDo_Type; (*Voltage middle position *) (*OldName:U_MIT;Cycle:5*)
		tU_Minus : HALioDo_Type; (*Voltage minus *) (*OldName:UMIN;Cycle:5*)
		tU_Plus : HALioDo_Type; (*Voltage plus *) (*OldName:UPLU;Cycle:5*)
		tOilSkid_PumpLP : HALioDo_Type; (*OilSkid low pressure pump (G.03-M-001)*) (*OldName:new pv;Cycle:5*)
		tOilSkid_PumpHP : HALioDo_Type; (*OilSkid high pressure pump (G.03-M-002)*) (*OldName:new pv;Cycle:5*)
		tOilSkid_PumpHP_UPS : HALioDo_Type; (*OilSkid high pressure pump - UPS (G.03-M-002)*) (*OldName:new pv;Cycle:5*)
		tOilSkid_PumpHP_Soft : HALioDo_Type; (*OilSkid high pressure pump - Soft (G.03-M-002)*) (*OldName:new pv;Cycle:5*)
		tOilSkid_PumpC : HALioDo_Type; (*OilSkid circulation pump (G.03-M-004)*) (*OldName:new pv;Cycle:5*)
		tOilSkid_Fan : HALioDo_Type; (*OilSkid fan*) (*OldName:new pv;Cycle:5*)
		tOilSkid_Heater : HALioDo_Type; (*OilSkid heater*) (*OldName:new pv;Cycle:5*)
		rPFSoll_lin_GC2GR : REAL; (*power factor setpoint GC->GR incl.GenReg.funct.1-7*) (*OldName:newPV;Cycle:5*)
		bP_Red_CosPCtr_U_Lo : BOOL; (*Power reduction by voltage low*) (*OldName:bPowRedGenSpgL;Cycle:5;*)
		bP_Red_CosPCtr_U_Hi : BOOL; (*Power reduction by voltage high*) (*OldName:bPowRedGenSpgH;Cycle:5;*)
		bP_Red_CosPCtr_F_Hi : BOOL; (*Power reduction by frequency high*) (*OldName:bPowRedGenFrqH;Cycle:5;*)
		bP_Red_CosPCtr_F_Lo : BOOL; (*Power reduction by frequnecy low*) (*OldName:bPowRedGenFrqL;Cycle:5;*)
		rPF_Lim_Norm : REAL; (*Generator power reduction due to Polar angle*) (*OldName:newpv;Cycle:5;*)
		rP_Red_CosPCtr_F_Norm : REAL; (*Generator power reduction due to Frequency*) (*OldName:ssPowerRedGenFrq;Cycle:5;*)
		rP_Red_CosPCtr_T_Norm : REAL; (*Generator power reduction due to Temperature*) (*OldName:ssPowerRedGenTemp;Cycle:5;*)
		rP_Red_CosPCtr_U_Norm : REAL; (*Generator power reduction due to Voltage*) (*OldName:ssPowerRedGenSpg;Cycle:5;*)
		rU_Gen_Exc : REAL; (*IF605 gen.excitation voltage*) (*OldName: ANA.ERREG; Cycle:5;*)
		bGCB_Off_CNS : BOOL; (*Generator circuit breaker opened by curent negative sequence*) (*OldName:gcb_off_iasy;Cycle:5*)
		bGCB_Off_RP : BOOL; (*Generator circuit breaker opened by reverse power*) (*OldName:gcb_off_rlsg;Cycle:5*)
		bPF_CosPCtr_block : BOOL; (*Block bit for generator controller*) (*OldName:Reg13_bBlock2;Cycle:5*)
		bU_Gen_match_isolated : BOOL; (*Speed related voltage adjustment active (local variable)*) (*OldName:u_adj_f_a;Cycle:5*)
		bU_SyD_match : BOOL; (*Voltage matching enabled*) (*OldName:dmnd_vmatch_synch;Cycle:5*)
		rPF_CosPCtr_block : REAL; (*Block value for generator controller*) (*OldName:Reg13_Block2;Cycle:5*)
		rPF_CosPCtr_Set_2 : REAL; (*NOT USED! power factor set point*) (*OldName:ssPF_STELL;Cycle:5*)
		rU_Gen_Mns_Set : REAL; (*Set mains voltage for PF- controller*) (*OldName:ssUnetzSoll;Cycle:5*)
		rCtrGenPF_Set : REAL; (*Generator ???*) (*OldName:new pv;Cycle:5*)
		rCtr_Q_Set : REAL; (*Generator Q controller*) (*OldName:new pv;Cycle:5*)
		rPF_AO_PF_I : REAL; (*power factor generator, mA signal*) (*OldName:AO_PF_gen_mA;Cycle:5*)
		rPF_AO_PF_U : REAL; (*power factor generator, V signal*) (*OldName:AO_PF_gen_V;Cycle:5*)
		bRelEngTurn_OilSkid : BOOL; (*release engine turn gear (Durchdrehvorrichtung) from Oil Skid*) (*OldName:new pv;Cycle:5*)
		bRelEngOp_OilSkid : BOOL; (*release engine operation from Oil Skid*) (*OldName:bRelEngOpGenLOS, rel_EngOp_LOS;Cycle:5*)
		rP_Red_T_GenAirIn_Norm : REAL; (*generator air inlet temperature power reduction*)
		tQ_AVR_Set_U : HALioAo_Type; (*reactive power setpoint for AlterantorVoltageRegulator V-Signal*) (*OldName:new pv;Cycle:5*)
		bMsg1036 : BOOL; (*overload short circuit*) (*OldName:new pv;Cycle:5*)
		bMsg1038 : BOOL; (*generator reverse power*) (*OldName:new pv;Cycle:5*)
		bMsg1073 : BOOL; (*generator over load from multi measuring device*) (*OldName:new pv;Cycle:5*)
		bMsg1132 : BOOL; (*generator differential protection*) (*OldName:new pv;Cycle:5*)
		bMsg1134 : BOOL; (*Earth failure*) (*OldName:new pv;Cycle:5*)
		bMsg3319 : BOOL; (*generator protection trip*) (*OldName:new pv;Cycle:5*)
		bRelEngStart_OilSkid : BOOL; (*release engine start from Oil Skid*) (*OldName:NewPv;Cycle:5*)
		rPF_Set_TimeTable : REAL; (*power factor setpoint from time table*) (*Oldname:newPv;Cycle:5;*)
		tU_Set_Norm : HALioAo_Type; (* voltage output for island mode [%Unom] *) (*OldName:new pv V4.07 ;Cycle:5*)
		bMsg1038Set : BOOL; (*Generator reverse power, Trip*)
		bMsg1109Set : BOOL; (*loss of excitation (trip)*)
		bMsg1110Set : BOOL; (*Generator frequency low, Trip*)
		bMsg1111Set : BOOL; (*Generator frequency high, Trip*)
		bMsg1112Set : BOOL; (*Neutral current high, Trip*)
		bMsg1126Set : BOOL; (*generator voltage low, Trip*)
		bMsg1127Set : BOOL; (*generator voltage high, Trip*)
		bMsg1143Set : BOOL; (*Voltage negative sequence (Voltage asymmetry), Trip*)
		bMsg1144Set : BOOL; (*Current negative sequnece (Current asymmetrt), Trip*)
		bMsg2277Set : BOOL; (*Generator voltage too low 2*)
		bMsg2316Set : BOOL; (*generator voltage high 2 (one phase)*)
		bAMM_OilSkid_PumpLP_CB : BOOL; (*Oilskid low pressure oil pump circuit breaker tripped*)
		bAMM_OilSkid_PumpHP_CB : BOOL; (*Oilskid high pressure oil pump circuit breaker tripped*)
		bAMM_OilSkid_MCB : BOOL; (*Oilskid main switch auxiliaries opened*)
		tCtr_Q_Out : _tGeACtrOut; (* Controller to visulization out structure *)
		bMsg9285 : BOOL; (*Measuring signal failure external voltage setpoint*)
		bPact_Rev : BOOL; (*Reverse power*)
		rP_Red_Eta_Gen_Norm : REAL; (*power reduction due to Cosphi<1 sent to OP [p.u.]*)
	END_STRUCT;
END_TYPE

(*END_OUT*)

TYPE
	Perm_GC_Struct : 	STRUCT
		iCnt_OilSkid_HP_PrErr : INT; (*synchronization operating mode selection*)
		iOpS_GndFailure : DINT; (*earth failure s*)
		iOpM_GndFailure : DINT; (*earth failure m*)
		iOpH_GndFailure : DINT; (*earth failure h*)
		rTB_PermValue04 : REAL; (*spare permanent value for testbench- replace with new vars of same lenght, when needed*) (*OldName:new PV;Cycle:2;*)
		rTB_PermValue05 : REAL; (*spare permanent value for testbench- replace with new vars of same lenght, when needed*) (*OldName:new PV;Cycle:2;*)
		rTB_PermValue06 : REAL; (*spare permanent value for testbench- replace with new vars of same lenght, when needed*) (*OldName:new PV;Cycle:2;*)
		rTB_PermValue07 : REAL; (*spare permanent value for testbench- replace with new vars of same lenght, when needed*) (*OldName:new PV;Cycle:2;*)
		rTB_PermValue08 : REAL; (*spare permanent value for testbench- replace with new vars of same lenght, when needed*) (*OldName:new PV;Cycle:2;*)
		rTB_PermValue09 : REAL; (*spare permanent value for testbench- replace with new vars of same lenght, when needed*) (*OldName:new PV;Cycle:2;*)
		rTB_PermValue10 : REAL; (*spare permanent value for testbench- replace with new vars of same lenght, when needed*) (*OldName:new PV;Cycle:2;*)
	END_STRUCT;
END_TYPE
```

### Module_GCPara.typ
```iecst
TYPE
	PROGRAMMER_INFO : 	STRUCT
		DO_NOT_SORT_PARA : STRING[40] := 'DO NOT CHANGE PARAMETER SORTING!'; (*DO NOT CHANGE PARAMETER SORTING!*) (*ADD NEW PARAMETER ONLY AT THE END OF THE Para STRUCTURE. DO NOT DELETE existing Para items.*)
	END_STRUCT;
	Para_GC_Struct : 	STRUCT
		rP_Act_LimLo : REAL; (*PARA [11509]: actual power low limit *) (*Oldname: GW_MS_PIST;Cycle:5*)
		bCtrGenPF_Active : BOOL; (*PARA [11485]: visibility generator controller*) (*Oldname:new pv;Cycle:5*)
		bGlowIgnPrevActive : BOOL; (*PARA [12089]: glow ignition prevention active*) (*Oldname:sel_GlowIgnPrevent;Cycle:5*)
		bPF_CosPCtr_Diff_Ena : BOOL; (*PARA [11486]: enable differential protection monitoring*) (*Oldname:DEAKT_DIFF;Cycle:5*)
		bPF_CosPCtr_Ena : BOOL; (*PARA [11487]: enable power factor controller on visualization*) (*Oldname:bQPF_XT;Cycle:5*)
		bPF_CosPCtr_F_Ena : BOOL; (*PARA [11488]: enable power reduction by generator frequency*) (*Oldname:bPowRed_GenFrq;Cycle:5*)
		bPF_CosPCtr_U_Ena : BOOL; (*PARA [11489]: enable power reduction by generator voltage*) (*Oldname:bPowRed_GenSpg;Cycle:5*)
		bT_Gen_Bear_A_Ena : BOOL; (*PARA [11490]: bearing A temperature monitoring enabled*) (*Oldname:lag1_a;Cycle:5*)
		bT_Gen_Bear_B_Ena : BOOL; (*PARA [11491]: bearing B temperature monitoring enabled*) (*Oldname:lag2_a;Cycle:5*)
		bT_Gen_Wind_Ena : BOOL; (*PARA [11492]: winding temperature monitoring enabled*) (*Oldname:wick_a;Cycle:5*)
		bU_Gen_Contr_Sel : BOOL; (*From settings task -> select fail safe DI_GENREG_F *) (*Oldname:sel_fs_DI_GENREG_F;Cycle:5*)
		bU_Gen_Exc_Ena : BOOL; (*PARA [11494]: excitation voltage monitoring enabled*) (*Oldname:u_erreg_a;Cycle:5*)
		bU_Gen_Mns_Match : BOOL; (*PARA [11495]: voltage matching active*) (*Oldname:vmatch_a;Cycle:5*)
		bU_Gen_P_Ena : BOOL; (*PARA [11496]: power related voltage adjustment active*) (*Oldname:u_adj_power_a;Cycle:5*)
		bU_Gen_spd_match : BOOL; (*PARA [11497]: speed related voltage adjustment active*) (*Oldname:u_adj_speed_a;Cycle:5*)
		iEng_Motortype : INT; (*Para: Motor type*) (*Oldname:iMotortyp;Cycle:5;*)
		rAng_CosPCtr_Lim : REAL; (*PARA [11501]: limit polar wheel angle for power factor controller*) (*Oldname:rDeltaPara;Cycle:5*)
		rAng_CosPCtr_Min : REAL; (*PARA [11502]: Minimum polar wheel angle for trip (LOSS OF EXCITATION)*) (*Oldname:rDelta_TripPara;Cycle:5*)
		rF_Gen_Match_Max : REAL; (*PARA [11503]: Generator frequency match maximum %Fnom*) (*Oldname:newPV;Cycle:5*)
		rF_Gen_Match_Min : REAL; (*PARA [11504]: Generator frequency match minmum %Fnom*) (*Oldname:newPV;Cycle:5*)
		rF_Nom : ARRAY[0..2]OF REAL; (*PARA [11736], [11737]: nominal generator frequency*) (*Oldname:usFreqNenn;Cycle:5*)
		rGen_CosPhi_Ena : REAL; (*PARA [11505]: Limit cos phi switching*) (*Oldname:GW_COS - calculated;Cycle:5*)
		rGen_CosPhi_Ena_Hy : REAL; (*PARA [11506]: Hysteresis cos phi switching*) (*Oldname:HY_COS;Cycle:5*)
		rN_EngNom : REAL; (*PARA [12128]: nominal speed*) (*Oldname:n_nenn;Cycle:5*)
		rN_EngStart_HyHi : REAL; (*PARA [11295]: speed engine start limit high hysteresis*) (*Oldname:HY_DREHZ;Cycle:5;*)
		rN_EngStart_HyHiHi : REAL; (*PARA [11507]: speed engine start limit high high hysteresis*) (*Oldname:HY_HDREHZ;Cycle:5*)
		rN_EngStart_LimHi : REAL; (*PARA [11296]: speed engine start limit high*) (*Oldname:GW_DREHZ;Cycle:5*)
		rN_EngStart_LimHiHi : REAL; (*PARA [11508]: speed engine start limit high high*) (*Oldname:GW_HDREHZ;Cycle:5*)
		rP_CosPCtr_F_Hi : REAL; (*PARA [11510]: minimum power at generator frequency high*) (*Oldname:ssPowRed_GenFrqHigh;Cycle:5*)
		rP_CosPCtr_F_Lo : REAL; (*PARA [11511]: minimum power at generator frequency low*) (*Oldname:ssPowRed_GenFrqLow;Cycle:5*)
		rP_CosPCtr_T_Hi : REAL; (*PARA [11512]: start power reduction winding temperature high*) (*Oldname:ssPowRed_GenWickHi;Cycle:5*)
		rP_CosPCtr_U_Hi : REAL; (*PARA [11513]: minimum power at generator voltage high*) (*Oldname:ssPowRed_GenVoltHigh;Cycle:5*)
		rP_CosPCtr_U_Lo : REAL; (*PARA [11514]: minimum power at generator voltage low*) (*Oldname:ssPowRed_GenVoltLow;Cycle:5*)
		rP_Reverse : REAL; (*PARA [11515]: reverse power limit*) (*Oldname:GW_RLSG;Cycle:5*)
		rP_Reverse_Hy : REAL; (*PARA [11516]: reverse power limit hysteresis*) (*Oldname:HY_RLSG;Cycle:5*)
		tiPF_CosPCtr_del : TIME; (*PARA [11620]: delay of reactive power monitoring*) (*Oldname:usReactDel[1] * 10;Cycle:5*)
		rPF_CosPCtr_F_Hi_End : REAL; (*PARA [11521]: power reduction ends at this generator (high) frequency value*) (*Oldname:ssGenFrqHighStop;Cycle:5*)
		rPF_CosPCtr_F_Hi_Start : REAL; (*PARA [11522]: power reduction starts at this generator (high) frequency value*) (*Oldname:ssGenFrqHighStart;Cycle:5*)
		rPF_CosPCtr_F_Lo_End : REAL; (*PARA [11523]: power reduction ends at this generator (low) frequency value*) (*Oldname:ssGenFrqLowStop;Cycle:5*)
		rPF_CosPCtr_F_Lo_Start : REAL; (*PARA [11524]: power reduction starts at this generator (low) frequency value*) (*Oldname:ssGenFrqLowStart;Cycle:5*)
		rPF_CosPCtr_F_ret : REAL; (*PARA [11525]: frequency value for retourning to normal power*) (*Oldname:ssFrqReturn;Cycle:5*)
		rPF_CosPCtr_h : ARRAY[0..5]OF REAL; (*PARA [11527], [11528], [11529], [11530], [11531]: map for time dependent power factor control*) (*Oldname:usPF_time_h;Cycle:5*)
		rPF_CosPCtr_m : ARRAY[0..5]OF REAL; (*PARA [11533], [11534], [11535], [11536], [11537]: map for time dependent power factor control*) (*Oldname:usPF_time_m;Cycle:5*)
		rPF_CosPCtr_T_max : REAL; (*PARA [11546]: maximum temp. For activation power factor reductions*) (*Oldname:twred_max;Cycle:5*)
		rPF_CosPCtr_T_red : REAL; (*PARA [11547]: gradient for power factor reduction by winding temperature high*) (*Oldname:twgradient;Cycle:5*)
		rPF_CosPCtr_T_wind : REAL; (*PARA [11548]: power reduction factor by generator winding temperature*) (*Oldname:wick_dp;Cycle:5*)
		rPF_CosPCtr_Tme_Set : ARRAY[0..5]OF REAL; (*PARA [11550], [11551], [11552], [11553], [11554]: power factor table for parameter entry time*) (*Oldname:rPF_Zeit;Cycle:5*)
		rPF_CosPCtr_U_Hi_End : REAL; (*PARA [11555]: power reduction ends at this generator (high) voltage value*) (*Oldname:ssGenVoltHighStop;Cycle:5*)
		rPF_CosPCtr_U_Hi_Start : REAL; (*PARA [11556]: power reduction starts at this generator (high) voltage value*) (*Oldname:ssGenVoltHighStart;Cycle:5*)
		rPF_CosPCtr_U_Lo_End : REAL; (*PARA [11557]: power reduction ends at this generator (low) voltage value*) (*Oldname:ssGenVoltLowStop;Cycle:5*)
		rPF_CosPCtr_U_Lo_Start : REAL; (*PARA [11558]: power reduction starts at this generator (low) voltage value*) (*Oldname:ssGenVoltLowStart;Cycle:5*)
		rS_Nom : REAL; (*PARA [11571]: Generator apparent nominal power*) (*Oldname:rS_CosP Ctr_act ;Cycle:5*)
		rT_Gen_Bear_Lim_A : REAL; (*PARA [11572]: generator bearing A temperature maximum, Warning*) (*Oldname:GW_LAGW1;Cycle:5*)
		rT_Gen_Bear_Lim_B : REAL; (*PARA [11573]: generator bearing B temperature maximum, Warning*) (*Oldname:GW_LAGW2;Cycle:5*)
		rT_Gen_Bear_Max_A : REAL; (*PARA [11574]: generator bearing A temperature maximum, Trip*) (*Oldname:GW_LAGA1;Cycle:5*)
		rT_Gen_Bear_Max_B : REAL; (*PARA [11575]: generator bearing B temperature maximum, Trip*) (*Oldname:GW_LAGA2;Cycle:5*)
		rT_Gen_Bear_Max_Hy_A : REAL; (*PARA [11576]: hysteresis generator bearing A temperature maximum*) (*Oldname:HY_LAG1;Cycle:5*)
		rT_Gen_Bear_Max_Hy_B : REAL; (*PARA [11577]: hysteresis generator bearing B temperature maximum*) (*Oldname:HY_LAG2;Cycle:5*)
		rT_Gen_Wind_Lim : REAL; (*PARA [11578]: Winding temperature maximum, Warning*) (*Oldname:GW_GWTW;Cycle:5*)
		rT_Gen_Wind_Lim_Hy : REAL; (*PARA [11579]: hysteresis generator winding temperature maximum*) (*Oldname:HY_GWTW;Cycle:5*)
		rT_Gen_Wind_Lim_Hy2 : REAL; (*PARA [11580]: hysteresis generator winding temperature maximum*) (*Oldname:HY_GWW;Cycle:5*)
		rT_Gen_Wind_Lim_L1 : REAL; (*PARA [11581]: generator winding temperature maximum phase 1, Warning*) (*Oldname:GW_GWW1;Cycle:5*)
		rT_Gen_Wind_Lim_L2 : REAL; (*PARA [11582]: generator winding temperature maximum phase 2, Warning*) (*Oldname:GW_GWW2;Cycle:5*)
		rT_Gen_Wind_Lim_L3 : REAL; (*PARA [11583]: generator winding temperature maximum phase 3, Warning*) (*Oldname:GW_GWW3;Cycle:5*)
		rT_Gen_Wind_Max : REAL; (*PARA [11584]: Winding temperature maximum, Trip*) (*Oldname:GW_GWTA;Cycle:5*)
		rT_Gen_Wind_Max_Hy : REAL; (*PARA [11585]: hysteresis generator winding temperature maximum*) (*Oldname:HY_GWA;Cycle:5*)
		rT_Gen_Wind_Max_Hy2 : REAL; (*PARA [11586]: hysteresis generator winding temperature maximum*) (*Oldname:HY_GWTA;Cycle:5*)
		rT_Gen_Wind_Max_L1 : REAL; (*PARA [11587]: generator winding temperature maximum phase 1, Trip*) (*Oldname:GW_GWA1;Cycle:5*)
		rT_Gen_Wind_Max_L2 : REAL; (*PARA [11588]: generator winding temperature maximum phase 2, Trip*) (*Oldname:GW_GWA2;Cycle:5*)
		rT_Gen_Wind_Max_L3 : REAL; (*PARA [11589]: generator winding temperature maximum phase 3, Trip*) (*Oldname:GW_GWA3;Cycle:5*)
		rU_Gen_Diff_Idle : REAL; (*PARA [11590]: voltage offset at idle operation %Un*) (*Oldname:U_offset_0PN;Cycle:5*)
		rU_Gen_Diff_Pn : REAL; (*PARA [11591]: voltage offset at full load %Un*) (*Oldname:U_offset_100PN;Cycle:5*)
		rU_Gen_ExcHi : REAL; (*PARA [11592]: excitation voltage high*) (*Oldname:GW_ERGW2;Cycle:5*)
		rU_Gen_ExcHyHi : REAL; (*PARA [11593]: excitation voltage high hysteresis*) (*Oldname:HY_ERGW2;Cycle:5*)
		rU_Gen_ExcHyLo : REAL; (*PARA [11594]: excitation voltage low hysteresis*) (*Oldname:HY_ERGW1;Cycle:5*)
		rU_Gen_ExcLo : REAL; (*PARA [11595]: excitation voltage low*) (*Oldname:GW_ERGW1;Cycle:5*)
		rU_Gen_match_delta : REAL; (*PARA [11596]: voltage matching per pulse %Unom/s*) (*Oldname:delta_u;Cycle:5*)
		rU_Gen_Nom : ARRAY[0..2]OF REAL; (*PARA [11597], [11598]: nominal voltage generator [70V..65kV]*) (*Oldname:usUNennGen;Cycle:5*)
		rU_Gen_Rmp_Dec : REAL; (*PARA [11600]: Maximum negative voltage adjustment ramp in %Unom/s*) (*Oldname:U_adj_ramp;Cycle:5*)
		rU_Gen_Rmp_Inc : REAL; (*PARA [11601]: Maximum positive voltage adjustment ramp in %Unom/s*) (*Oldname:U_adj_ramp;Cycle:5*)
		rU_adj_max_up : REAL; (*PARA [12438]: Maximum positive voltage adjustment in %Unom*) (*Oldname: U_adj_max_up; Cycle: 5*)
		rU_adj_max_down : REAL; (*PARA [12439]: Maximum negative voltage adjustment in %Unom*) (*Oldname: U_adj_max_down; Cycle: 5*)
		rU_SyncNom : ARRAY[0..2]OF REAL; (*PARA [11859], [11860]: nominal voltage sync1 & sync2 [70V..65kV]*) (*Oldname:usUNennSync;Cycle:5*)
		rxd_CosPCtr : REAL; (*PARA [11602]: Synchronous reactance xd*) (*Oldname:r_xd;Cycle:5*)
		tCtrGenPF : _tGeACtrPara; (*Para controller Generator*) (*Oldname:new pv;Cycle:5*)
		ti_Gen_VoltReg_Fail : TIME; (*PARA [11616]: timer generator voltage regulator failure (Standard =T#0s ; Basler = T#60s)*) (*Oldname:new pv; Cycle:5*)
		tiP_Gen_Reverse : TIME; (*PARA [11617]: timer (10 sec) for delay after gen. Circuit breaker closed*) (*Oldname:TW_AT24;Cycle:5*)
		tiP_Gen_Reverse2 : TIME; (*PARA [11618]: timer (10 sec) for delay of generator reverse power*) (*Oldname:TW_T28;Cycle:5*)
		tiP_Reverse_Mon_Ena : TIME; (*PARA [11619]: timer (10 sec) for activation monitoring reverse power *) (*Oldname:TW_RLSG_W;Cycle:5*)
		bU_adj_gcb_ext_hilo_a : BOOL; (*PARA [12442]: voltage adjust for GCB sync. external Hi/Low enable*) (*Oldname:u_adj_gcb_ext_hilo_a;Cycle:5;*)
		bU_adj_gcb_mmd_calc_a : BOOL; (*PARA [12440]: voltage adjust for GCB sync. MMD calc enable*) (*Oldname:u_adj_gcb_mmd_calc_a;Cycle:5;*)
		bU_adj_mcb_ext_hilo_a : BOOL; (*PARA [12443]: voltage adjust for MCB sync. external Hi/Low enable*) (*Oldname:u_adj_mcb_ext_hilo_a;Cycle:5;*)
		bU_adj_mcb_mmd_calc_a : BOOL; (*PARA [12441]: voltage adjust for MCB sync. MMD calc enable*) (*Oldname:u_adj_mcb_mmd_calc_a;Cycle:5;*)
		rTi_Q_MinDel : ARRAY[0..2]OF REAL; (*PARA [11835], [11836]: delay reactive power monitoring *) (*OldName:usReactDel; Cycle: *)
		bSyActive : BOOL; (*PARA [12195]: synchronization functions active *) (*OldName:bSynch; Cycle:5;*)
		bOilSkid_Exist : BOOL; (*PARA [12528]: OilSkid active	*) (*Oldname:new pv; Cycle:5*)
		bFlow_OilSkid_DE_Exist : BOOL; (*PARA [12543]: Oil flow to DE storage active	*) (*Oldname:new pv; Cycle:5*)
		bFlow_OilSkid_NDE_Exist : BOOL; (*PARA [12548]: Oil flow to NDE storage activ	*) (*Oldname:new pv; Cycle:5*)
		bLev_OilSkid_Tank_Exist : BOOL; (*PARA [12529]: Oil tank level active	*) (*Oldname:new pv; Cycle:5*)
		bPr_OilSkid_HP_DE_Exist : BOOL; (*PARA [12557]: Oil pressure in high pressure circle to DE Storage active	*) (*Oldname:new pv; Cycle:5*)
		bPr_OilSkid_HP_NDE_Exist : BOOL; (*PARA [12558]: Oil pressure in high pressure circle to NDE Storage active	*) (*Oldname:new pv; Cycle:5*)
		bT_OilSkid_Supply_Exist : BOOL; (*PARA [12538]: Oil pre-temperaure active (�lvorlauftemperatur) 	*) (*Oldname:new pv; Cycle:5*)
		bT_OilSkid_Tank_Exist : BOOL; (*PARA [12534]: Oil tank temperature activ	*) (*Oldname:new pv; Cycle:5*)
		rFlow_OilSkid_DE_Hi : REAL; (*PARA [12547]: Oil flow to DE storage Maximum - Warning [l/min]*) (*Oldname:new pv; Cycle:5*)
		rFlow_OilSkid_DE_Lo : REAL; (*PARA [12546]: Oil flow to DE storage Minimum - Warning [l/min]*) (*Oldname:new pv; Cycle:5*)
		rFlow_OilSkid_NDE_Hi : REAL; (*PARA [12552]: Oil flow to NDE storage Maximum- Warning [l/min]*) (*Oldname:new pv; Cycle:5*)
		rFlow_OilSkid_NDE_Lo : REAL; (*PARA [12551]: Oil flow to NDE storage Minimum - Warning [l/min]*) (*Oldname:new pv; Cycle:5*)
		rLev_OilSkid_Tank_Lo : REAL; (*PARA [12532]: Oil tank level  Minimum - Warning [%]*) (*Oldname:new pv; Cycle:5*)
		rLev_OilSkid_Tank_LoLo : REAL; (*PARA [12533]: Oil tank level Minimum - Error [%]*) (*Oldname:new pv; Cycle:5*)
		rPr_OilSkid_HP_Lo : REAL; (*PARA [12556]: Oil pressure in high pressure circle Minimum � Warning [bar]*) (*Oldname:new pv; Cycle:5*)
		rT_OilSkid_Supply_Hi : REAL; (*PARA [12542]: Oil pre-temperaure active Maximum - Warning [°C]*) (*Oldname:new pv; Cycle:5*)
		rT_OilSkid_Supply_Lo : REAL; (*PARA [12541]: Oil pre-temperaure active Minimum - Warning [°C]*) (*Oldname:new pv; Cycle:5*)
		rT_OilSkid_Tank_Set : REAL; (*PARA [12537]: Oil tank set temperature [°C]*) (*Oldname:new pv; Cycle:5*)
		tiOilSkid_PumpHP_Run : TIME; (*PARA [12553]: Time untill the high pressure pump switched off [s]*) (*Oldname:new pv; Cycle:5*)
		bF_GenBear_DE1_Active : BOOL; (*PARA [12706]: vibration generator bearing drive end 1 measuring signal activ*) (*Oldname:v_GenBear_a;Cycle:5;*)
		bF_GenBear_DE2_Active : BOOL; (*PARA [12707]: vibration generator bearing drive end 2 measuring signal activ*) (*Oldname:v_GenBear_a;Cycle:5;*)
		bF_GenBear_NDE1_Active : BOOL; (*PARA [12708]: vibration generator bearing non drive end 1 measuring signal activ*) (*Oldname:v_GenBear_a;Cycle:5;*)
		bF_GenBear_NDE2_Active : BOOL; (*PARA [12709]: vibration generator bearing non drive end 2 measuring signal activ*) (*Oldname:v_GenBear_a;Cycle:5;*)
		rF_GenBear_Hi : REAL; (*PARA [12712]: vibration generator bearing limit high*) (*Oldname:GW_v_GenBear_hi2;Cycle:5;*)
		tiF_GenBear_Hi : TIME; (*PARA [12713]: delay bearing displacement high*) (*Oldname:TW_v_GenBear_hi2;Cycle:5*)
		rF_GenBear_HiHi : REAL; (*PARA [12714]: vibration generator bearing limit high high*) (*Oldname:GW_v_GenBear_hi2;Cycle:5;*)
		tiF_GenBear_HiHi : TIME; (*PARA [12717]: delay bearing displacement high high*) (*Oldname:TW_v_GenBear_hi2;Cycle:5*)
		bT_GenAirIn_Active : BOOL; (*PARA [12715]: generator air inlet temperature measuring signal activ*) (*Oldname:t_GenAirIn_a;Cycle:5;*)
		bT_GenAirOut_Active : BOOL; (*PARA [12716]: generator air outlet temperature measuring signal activ*) (*Oldname:t_GenAirOut_a;Cycle:5;*)
		bT_GenAirIn2_Active : BOOL; (*PARA [13695]: generator air inlet temperature 2 measuring signal activ*) (*Oldname:newPv;Cycle:5;*)
		rT_Pred_GenAirIn_Start : REAL; (*PARA [13696]: generator air inlet temperature start power reduction*) (*Oldname:newPv;Cycle:5;*)
		rT_Pred_GenAirIn_Rate : REAL; (*PARA [13697]: generator air inlet temperature rate power reduction*) (*Oldname:newPv;Cycle:5;*)
		rQ_UnderExc_Lim : REAL; (*PARA [13693]: reactive power limit underexcitated [%]*) (*Oldname:newPv;Cycle:5;*)
		rQ_OverExc_Lim : REAL; (*PARA [13694]: reactive power limit overexcitated [%]*) (*Oldname:newPv;Cycle:5;*)
		bCtr_Q : BOOL; (*PARA [14107]: visibility generator Q controller*) (*Oldname:newPv;Cycle:5*)
		tCtr_Q : _tGeACtrPara; (*Para generator Q controller*) (*Oldname:newPv;Cycle:5*)
		iQ_GrC_PointCtrl : INT; (*PARA [13992]: Q controller - selection point of control*) (*Oldname:newPv;Cycle:5;*)
		rU_GrC_SetEU_Nom : REAL; (*PARA [11696]: [V] Nominal voltage for voltage setpoint *) (* OldName: ulUnom_evu; Cycle: 5 *)
		iQ_GrC_CtrlFun : USINT; (*PARA [13991]: select Q/PF control function: 0:custom 1:PFset 2:PF(P) 3:PF(U) 4:Q(U) 5:Q(P) 6:Qset 7:Uset 8:time table*)
		rV_Over2 : ARRAY[0..2]OF REAL; (*Para: over voltage 2[V]*) (*Oldname:newPv;Cycle:5;*)
		rTi_V_Over2 : ARRAY[0..2]OF REAL; (*Para: over voltage 2 delay*) (*Oldname:newPv;Cycle:5;*)
		bQ_UnderExc_Ena : BOOL; (*PARA [14284]: Reactive power reduction by voltage enabled*)
		rQ_UnderExc_Start : REAL; (*PARA [14285]: Start value low voltage (Umin1)*)
		rQ_UnderExc_Stop : REAL; (*PARA [14286]: Stop value low voltage (Umin2)*)
		rQ_UnderExc_Lim2 : REAL; (*PARA [14287]: Reduced reactive power low voltage(Qlim2)*)
		iSource_U_OffsSet : INT; (*PARA [14298]: Voltage offset set point in island mode: 0= no setpoint, 1= Droop, 2= External *)
		rU_StCtr_Grad : REAL; (*PARA [14299]: Gradient for the voltage droop curve in island mode [%Unom]*)
		rEta_Gen_PF1 : REAL; (*PARA [14343]: Generator Efficiency at power factor 1.0*)
		rEta_Gen_PF08 : REAL; (*PARA [14344]: Generator Efficiency at power factor 0.8 overexcited*)
		iU_Isl_SetX : INT; (*PARA [14705]: choice of voltage setpoint: 0=not used, 1=Internal Setpoint, 2=Voltage backup set point; 3=External Bus, 4=Customized, 5=External AI*)
		rU_Isl_SetInt : REAL; (*PARA [14706]: voltage internal setpoint*)
		rU_SetExtAI_SetI1 : REAL; (*PARA [14707]: voltage external setpoint AI, current point 1*)
		rU_SetExtAI_SetI2 : REAL; (*PARA [14708]: voltage external setpoint AI, current point 2*)
		rU_SetExtAI_SetP1 : REAL; (*PARA [14709]: voltage external setpoint AI, voltage point 1*)
		rU_SetExtAI_SetP2 : REAL; (*PARA [14710]: voltage external setpoint AI, voltage point 2*)
		rU_Isl_SetAct_BU : REAL; (*PARA [14711]: voltage external setpoint, backup value*)
		bRelFreeze_Uset_Isl : BOOL; (*PARA [14712]: voltage external setpoint, interruption characteristic: 0=backup value, 1=last valid value*)
		iQ_Droop_SetX : INT; (*PARA [14713]: choice of reactive power setpoint: 0=not used, 1=Internal Setpoint, 2=Voltage backup set point; 3=External Bus, 4=Customized, 5=External AI*)
		rQ_Droop_SetInt : REAL; (*PARA [14714]: reactive power internal setpoint, -x[underexcited]/+x[overexcited]*)
		rQ_Droop_Set_SetI1 : REAL; (*PARA [14715]: reactive power external setpoint AI, current point 1*)
		rQ_Droop_Set_SetI2 : REAL; (*PARA [14716]: reactive power external setpoint AI, current point 2*)
		rQ_Droop_Set_SetP1 : REAL; (*PARA [14717]: reactive power external setpoint AI, reactive power point 1, -x[underexcited]/+x[overexcited]*)
		rQ_Droop_Set_SetP2 : REAL; (*PARA [14718]: reactive power external setpoint AI, reactive power point 2, -x[underexcited]/+x[overexcited]*)
		rQ_Droop_SetAct_BU : REAL; (*PARA [14719]: reactive power external setpoint, backup value, -x[underexcited]/+x[overexcited]*)
		bRelFreeze_Qset_Droop : BOOL; (*PARA [14720]: reactive power external setpoint, interruption characteristic: 0=backup value, 1=last valid value*)
		bComm1_Ena : BOOL; (*PARA [10165]: link 1 release data receive enabled*) (*OldName:Kopl1Empf; Cycle: 5;*)
		bComm2_Ena : BOOL; (*PARA [10166]: link 2 release data receive enabled*) (*OldName:Kopl2Empf; Cycle: 5;*)
		bMMDGroundFaultMonAct : BOOL;(*PARA [14943]: Earth fault monitoring via MMU signals activated*)
		tTi_MMDGroundFaultWarning : TIME; (*PARA [14944]: delay MMD earth fault warning*)
		tTi_MMDGroundFaultTrip : TIME; (*PARA [14945]: delay MMD earth fault trip*)
		bCAsym_Ena : BOOL; (*PARA [15070]: Enable unbalance current monitoring*)
	END_STRUCT;
END_TYPE
```

### module_GC.var
```iecst
VAR
	VIS2MM : VIS2MM_Struct;
	IN_GC : IN_GC_Struct;
	MM2VIS : MM2VIS_Struct;
	OUT_GC : OUT_GC_Struct;
	Para : Para_GC_Struct;
	ParaFactoryDefault : Para_GC_Struct;
	pm : Para_GC_Struct;
	tCtrGenPF_In : _tGeACtrIn;
	tCtrGenPF_Out : _tGeACtrOut;
	xCtrGenPF : GeACtr;
	xEngType : EngType; (*Engine type defintion*)
	xOpMode : OpMode;
	PF_Ist_lin : REAL;
	PFSoll_lin : REAL;
	bOMSS_Scav : BOOL; (*Operation mode selector switch - Scavenging*)
	bOMSS_MAT : BOOL; (*Operation mode selector switch - Manual automatic*)
	bOMSS_Test : BOOL; (*Operation mode selector switch - Test*)
	bOMSS_Aut : BOOL; (*Operation mode selector switch - Auto*)
	bOMSS_Man : BOOL; (*Operation mode selector switch - Manual*)
	bGnlTrip1 : BOOL; (*general trip *)
	bGnlTrip2 : BOOL; (*general trip *)
	bGnlTrip3 : BOOL; (*general trip *)
	bGnlTrip : BOOL; (*general trip *)
	bGnlWarning : BOOL; (*general warning*)
	M_DREHZ : BOOL; (*Engine starter speed exceeded*)
	M_HDREHZ : BOOL; (*Engine speed start limit high*)
	bEng_Run_10s : BOOL; (*Engine in operation since 10 seconds*)
	bEng_Run_20s : BOOL; (*Engine in operation since 20 seconds*)
	bGen_CosPhi_Ena : BOOL; (*Old name AN_COS*)
	bMI_MMU : BOOL; (*mains import measurement by MMU*)
	bMIPCont : BOOL; (*mains import power controller active*)
	bMIPCont_SPext : BOOL; (*ext. set point of mains power control active*)
	bMIRPCont_SPext : BOOL; (*ext. set point for mains import react. pow. active*)
	bPF_CosPCtr_Trip : BOOL;
	bPF_LIM_Temp : BOOL; (*PF limitation by alternator winding temp.*)
	bT_Gen_Bear_A_Lim : BOOL;
	bT_Gen_Bear_A_Max : BOOL;
	bT_Gen_Bear_B_Lim : BOOL;
	bT_Gen_Bear_B_Max : BOOL;
	bT_Gen_Wind_L1_Lim : BOOL;
	bT_Gen_Wind_L1_Max : BOOL;
	bT_Gen_Wind_L2_Lim : BOOL;
	bT_Gen_Wind_L2_Max : BOOL;
	bT_Gen_Wind_L3_Lim : BOOL;
	bT_Gen_Wind_L3_Max : BOOL;
	bT_Gen_Wind_Lim : BOOL;
	bT_Gen_Wind_Max : BOOL;
	bU_Gen_Exc_Max : BOOL;
	bU_Gen_Exc_Min : BOOL;
	PF_1_fix : REAL := 0.0;
	PF_2_fix : REAL := 0.0;
	PF_Out1 : INT;
	PF_Out2 : INT;
	rAng_CosPCtr_LimCalc : REAL;
	rAng_CosPCtr_MinCalc : REAL;
	rP_CosPCtr_F_Red : REAL; (*power reduction due to high or low frequency*)
	rP_CosPCtr_T_Red : REAL; (*power reduction due to high winding temperature*)
	rP_CosPCtr_U_Red : REAL; (*power reduction due to high or low voltage*)
	rP_Gen_ppt : REAL;
	rPF_CosPCtr_LimCalc1 : REAL;
	rPF_CosPCtr_LimCalc2 : REAL;
	rPF_CosPCtr_MinCalc1 : REAL;
	rPF_CosPCtr_MinCalc2 : REAL;
	rPF_CosPCtr_Set_Ctr13 : REAL;
	rQ_CosPCtr_Set : REAL;
	rU_AI_Gen_Avg_ppt : REAL;
	ssMIPCont_SP : INT; (*set point of mains power control*)
	ssMIRPCont_SP : INT; (*set point of mains reactive power control*)
	ssP_mains_scale1 : INT; (*scaling of mains power at 4mA*)
	ssP_mains_scale2 : INT; (*scaling of mains power at 20mA*)
	ssQ_mains_scale1 : INT; (*scaling of mains reactive power at 4mA*)
	ssQ_mains_scale2 : INT; (*scaling of mains reactive power at 20mA*)
	ssQ_mainsOffset : INT; (*offset value for mains reactive power controller*)
	U_fix : REAL := 0.0;
	rU_Gen_Diff_Match_I : REAL; (*voltage offset for power factor controller, current signal (mA)*)
	rU_Gen_Diff_Match_U : REAL; (*voltage offset for power factor controller, voltage signal (V)*)
	bNoInitDetected : BOOL := FALSE; (*allways true, except 1cycle on init up*)
	rU_Gen_f_match : REAL; (*Frequency related voltage adjustment value*) (*OldName:u_offset_f_r;Cycle:5*)
	rU_Gen_sy_match : REAL; (*Voltage offset for voltage matching during synchr.*) (*OldName:u_offset_sy_r;Cycle:5*)
	rU_Gen_P_match : REAL; (*Power related voltage adjustment value*) (*OldName:u_offset_p_r;Cycle:5*)
	bU_minus_MMU : BOOL;
	bU_plus_MMU : BOOL;
	bU_Gen_P_match : BOOL; (*Power related voltage adjustment active*) (*OldName:u_adj_p_a;Cycle:5*)
	bMsg2156 : BOOL; (*Q-RED by winding temperature limit*) (*OldName:RPSDIA[35];Cycle:5*)
	bMsg2157 : BOOL; (*Q-limit by polar wheel angle*) (*OldName:RPSDIA[36];Cycle:5*)
	bAMM_Lev_OilSkid_Sump_Hi : BOOL := FALSE; (*W3418 Oilskid oil in oil sump *)
	bAMM_Lev_OilSkid_Tank_Ms : BOOL := FALSE; (*W3419 Oilskid tank oil level measuring signal failure *)
	bAMM_Lev_OilSkid_Tank_Lo : BOOL := FALSE; (*W3420 Oilskid tank oil level low*)
	bAMM_Lev_OilSkid_Tank_LoLo : BOOL := FALSE; (*A2208 Oilskid tank oil level low *)
	bAMM_T_OilSkid_Tank_Ms : BOOL := FALSE; (*W3421 Oilskid tank oil temperature measuring signal failure*)
	bAMM_T_OilSkid_Tank_Lo : BOOL := FALSE; (*W3422 Oilskid tank oil temperature low*)
	bAMM_T_OilSkid_Supply_Ms : BOOL := FALSE; (*W3423 Oilskid oil supply temperature measuring signal failure*)
	bAMM_T_OilSkid_Supply_Lo : BOOL := FALSE; (*W3424 Oilskid oil supply temperature low*)
	bAMM_T_OilSkid_Supply_Hi : BOOL := FALSE; (*W3425 Oilskid oil supply temperature high*)
	bAMM_OilSkid_PumpLP_CB : BOOL := FALSE; (*W3426 Oilskid low pressure oil pump circuit breaker tripped*)
	bAMM_Flow_OilSkid_DE_Ms : BOOL := FALSE; (*W3427 Oilskid oil flow TO DE bearing measuring signal failure*)
	bAMM_Flow_OilSkid_DE_Lo : BOOL := FALSE; (*W3428 Oilskid oil flow TO DE bearing low*)
	bAMM_Flow_OilSkid_DE_Hi : BOOL := FALSE; (*W3429 Oilskid oil flow TO DE bearing high*)
	bAMM_Flow_OilSkid_NDE_Ms : BOOL := FALSE; (*W3430 Oilskid oil flow TO NDE bearing measuring signal failure*)
	bAMM_Flow_OilSkid_NDE_Lo : BOOL := FALSE; (*W3431 Oilskid oil flow TO NDE bearing low*)
	bAMM_Flow_OilSkid_NDE_Hi : BOOL := FALSE; (*W3432 Oilskid oil flow TO NDE bearing high*)
	bAMM_DPr_OilSkid_FiltLP_Hi : BOOL := FALSE; (*W2505 Oilskid low pressure oil filter clogged*)
	bAMM_OilSkid_PumpHP_CB : BOOL := FALSE; (*W3433 Oilskid high pressure oil pump circuit breaker tripped*)
	bAMM_OilSkid_PumpHP_CB_UPS : BOOL := FALSE; (*W3434 Oilskid high pressure oil pump circuit breaker tripped - UPS*)
	bAMM_Pr_OilSkid_HP_DE_Ms : BOOL := FALSE; (*W3435 Oilskid oil pressure TO DE bearing measuring signal failure*)
	bAMM_Pr_OilSkid_HP_DE_Lo : BOOL := FALSE; (*W3436 Oilskid oil pressure TO DE bearing low*)
	bAMM_Pr_OilSkid_HP_NDE_Ms : BOOL := FALSE; (*W3442 Oilskid oil pressure TO NDE bearing measuring signal failure*)
	bAMM_Pr_OilSkid_HP_NDE_Lo : BOOL := FALSE; (*W3443 Oilskid oil pressure TO NDE bearing low*)
	bAMM_DPr_OilSkid_FiltHP_DE_Hi : BOOL := FALSE; (*W2508 Oilskid high pressure oil filter DE clogged*)
	bAMM_DPr_OilSkid_FiltHP_NDE_Hi : BOOL := FALSE; (*W3446 Oilskid high pressure oil filter NDE clogged*)
	bAMM_OilSkid_Fan_CB : BOOL := FALSE; (*W3437 Oilskid fan circuit breaker tripped*)
	bAMM_OilSkid_Heater_CB : BOOL := FALSE; (*W3438 Oilskid heater circuit breaker tripped*)
	bAMM_OilSkid_MCB : BOOL := FALSE; (*W3439 Oilskid main switch auxiliaries opened*)
	bAMM_OilSkid_AuxV : BOOL := FALSE; (*W3440 Oilskid auxiliaries voltage NOT available*)
	bAMM_OilSkid_AuxV_UPS : BOOL := FALSE; (*W3441 Oilskid auxiliaries voltage NOT available - UPS*)
	bAMM_OilSkid_PumpC_CB : BOOL := FALSE; (*W3447 Oilskid circulation pump circuit breaker tripped *)
	bN_EngAct_IsZero : BOOL := FALSE; (*Actual speed [1/min] is Zero *)
	bEng_Run_30m : BOOL := FALSE; (*Engine operation + 30 minutes*)
	bMsg2208_Test : BOOL; (*Prio3: oilskid tank level minimum - TEST*)
	rPF_POC_Act : REAL;
	tCtr_Q_In : _tGeACtrIn;
	tCtr_Q_Out : _tGeACtrOut;
	xCtr_Q : GeACtr;
	rS_POC_Act : REAL; (*aparent power at selected point of control [kVA]*)
	rP_POC_Act : REAL; (*active power at selected point of control [kW]*)
	rQ_POC_Act : REAL; (*reactive power at selected point of control [kVAr]*)
	rU_POC_Act : REAL; (*average vooltage at selected point of control [V]*)
	rS_POC_Act_Norm : REAL; (*aparent power at selected point of control [%]*)
	rP_POC_Act_Norm : REAL; (*active power at selected point of control [%]*)
	rQ_POC_Act_Norm : REAL; (*reactive power at selected point of control [%]*)
	rQ_POC_Act_CalcV : REAL; (*reactive power at selected point of control calculated from voltage [%]*)
	rQ_Set_Lim : REAL; (*reactive power setpoint limited*)
	rQ_Set_Sum : REAL; (*reactive power setpoint limited summary*)
	rU_Gen_Diff_Match : REAL; (*calc.setpoint offset from v_ctr *)
	bMsg9351 : BOOL; (*Measuring signal failure external reactive power set point for voltage droop mode*)
	bMsg9285 : BOOL; (*Measuring signal failure external voltage setpoint*)
	bMsg2998 : BOOL; (*Q-limit by under voltage*)
	iOpS_GndFailure : DINT; (*earth failure s*)
	iOpM_GndFailure : DINT; (*earth failure m*)
	tiGoodQual : TIME := T#5s; (*Time for signal Quality check*)
	bRelMon_Flow_DE : BOOL := FALSE; (*Release monitoring OilSkid oil flow to DE*)
	bRelMon_Flow_NDE : BOOL := FALSE; (*Release monitoring OilSkid oil flow to NDE*)
	bMsg9372_set : BOOL; (*W9372 Multi measurement device: Earth failure generator*)
	bMsg2373_set : BOOL; (*A2373 Multi measurement device: Earth failure generator*)
END_VAR
```

### Program Logical/Generator/defaultGC (IEC, version 4.12.0) - default

#### defaultGCCyclic.st
```iecst
(*******************************************************************************
default		value set

This code is confidential and proprietary to the INNIO Company.
It may not be used in any form, or reproduced in any manner,
without the express written permission of the INNIO Company.
Copyright, INNIO Company, 2022

Customized modifications: -
------------------------

History:
-------
V0.00.0	21.11.2012	Ganguly.		new
V3.99.0	11.03.2013	lettenbichler	preset for tGen_LO_CoolingSys_Fail added
									preset for tU_Gen_LimLo2[1] added
V4.00.0 28.01.2015	lettenb.		920 added(stapelfeld)
V4.03.0	22.07.2015	lettenb.		dyn.gridcode III(thaler)
V4.09.0	02.12.2019	lettenb.		ground fault warning added(thaler)
V4.12.0	21.11.2022	lettenb.		automatic generator greasing system

 ********************************************************************)

PROGRAM _CYCLIC

	(* default TRUE setting for not existing Di's *)
	IN_GC.tOlShortCirc.Di      			:=  IN_GC.tOlShortCirc.Di 				OR NOT IN_GC.tOlShortCirc.GoodQual;
	IN_GC.tF_MMD_LimHi[0].Di      		:=  IN_GC.tF_MMD_LimHi[0].Di 			OR NOT IN_GC.tF_MMD_LimHi[0].GoodQual;
	IN_GC.tF_MMD_LimHi[1].Di       		:=  IN_GC.tF_MMD_LimHi[1].Di 			OR NOT IN_GC.tF_MMD_LimHi[1].GoodQual;
	IN_GC.tF_MMD_LimHi[2].Di       		:=  IN_GC.tF_MMD_LimHi[2].Di 			OR NOT IN_GC.tF_MMD_LimHi[2].GoodQual;
	IN_GC.tF_MMD_LimLo[0].Di       		:=  IN_GC.tF_MMD_LimLo[0].Di 			OR NOT IN_GC.tF_MMD_LimLo[0].GoodQual;
	IN_GC.tF_MMD_LimLo[1].Di       		:=  IN_GC.tF_MMD_LimLo[1].Di 			OR NOT IN_GC.tF_MMD_LimLo[1].GoodQual;
	IN_GC.tF_MMD_LimLo[2].Di      		:=  IN_GC.tF_MMD_LimLo[2].Di 			OR NOT IN_GC.tF_MMD_LimLo[2].GoodQual;
	IN_GC.tI_MMD_Neutr_LimHi[0].Di 		:=  IN_GC.tI_MMD_Neutr_LimHi[0].Di 		OR NOT IN_GC.tI_MMD_Neutr_LimHi[0].GoodQual;
	IN_GC.tI_MMD_Neutr_LimHi[1].Di 		:=  IN_GC.tI_MMD_Neutr_LimHi[1].Di 		OR NOT IN_GC.tI_MMD_Neutr_LimHi[1].GoodQual;
	IN_GC.tI_MMD_Neutr_LimHi[2].Di 		:=  IN_GC.tI_MMD_Neutr_LimHi[2].Di 		OR NOT IN_GC.tI_MMD_Neutr_LimHi[2].GoodQual;
	IN_GC.tU_Gen_LimLo[0].Di       		:=  IN_GC.tU_Gen_LimLo[0].Di 			OR NOT IN_GC.tU_Gen_LimLo[0].GoodQual;
	IN_GC.tU_Gen_LimLo[1].Di       		:=  IN_GC.tU_Gen_LimLo[1].Di 			OR NOT IN_GC.tU_Gen_LimLo[1].GoodQual;
	IN_GC.tU_Gen_LimLo[2].Di       		:=  IN_GC.tU_Gen_LimLo[2].Di 			OR NOT IN_GC.tU_Gen_LimLo[2].GoodQual;
	IN_GC.tU_Gen_LimHi[0].Di       		:=  IN_GC.tU_Gen_LimHi[0].Di 			OR NOT IN_GC.tU_Gen_LimHi[0].GoodQual;
	IN_GC.tU_Gen_LimHi[1].Di       		:=  IN_GC.tU_Gen_LimHi[1].Di 			OR NOT IN_GC.tU_Gen_LimHi[1].GoodQual;
	IN_GC.tU_Gen_LimHi[2].Di       		:=  IN_GC.tU_Gen_LimHi[2].Di 			OR NOT IN_GC.tU_Gen_LimHi[2].GoodQual;

	IN_GC.tU_Gen_LimLo2[1].Di			:=	IN_GC.tU_Gen_LimLo2[1].Di			OR NOT IN_GC.tU_Gen_LimLo2[1].GoodQual;
	IN_GC.tI_MMD_Asy[0].Di				:=  IN_GC.tI_MMD_Asy[0].Di 				OR NOT IN_GC.tI_MMD_Asy[0].GoodQual;
	IN_GC.tI_MMD_Asy[1].Di				:=  IN_GC.tI_MMD_Asy[1].Di				OR NOT IN_GC.tI_MMD_Asy[1].GoodQual;
	IN_GC.tI_MMD_Asy[2].Di				:=  IN_GC.tI_MMD_Asy[2].Di				OR NOT IN_GC.tI_MMD_Asy[2].GoodQual;
	IN_GC.tU_MMD_Asy[0].Di				:=  IN_GC.tU_MMD_Asy[0].Di				OR NOT IN_GC.tU_MMD_Asy[0].GoodQual;
	IN_GC.tU_MMD_Asy[1].Di				:=  IN_GC.tU_MMD_Asy[1].Di				OR NOT IN_GC.tU_MMD_Asy[1].GoodQual;
	IN_GC.tU_MMD_Asy[2].Di				:=  IN_GC.tU_MMD_Asy[2].Di				OR NOT IN_GC.tU_MMD_Asy[2].GoodQual;
	IN_GC.tI_Diff.Di               		:=  IN_GC.tI_Diff.Di 					OR NOT IN_GC.tI_Diff.GoodQual;
	IN_GC.tU_GenOverVolt.Di       		:=  IN_GC.tU_GenOverVolt.Di 			OR NOT IN_GC.tU_GenOverVolt.GoodQual;
	IN_GC.tFlow_Gen_Lube.Di        		:=  IN_GC.tFlow_Gen_Lube.Di 			OR NOT IN_GC.tFlow_Gen_Lube.GoodQual;
	IN_GC.tI_MMD_LimHi.Di          		:=  IN_GC.tI_MMD_LimHi.Di 				OR NOT IN_GC.tI_MMD_LimHi.GoodQual;
	IN_GC.tDiffPrct.Di         			:=  IN_GC.tDiffPrct.Di					OR NOT IN_GC.tDiffPrct.GoodQual;
	IN_GC.tGndFailure.Di       			:=  IN_GC.tGndFailure.Di				OR NOT IN_GC.tGndFailure.GoodQual;
	IN_GC.tGenPrctTrip.Di     	 		:=  IN_GC.tGenPrctTrip.Di 				OR NOT IN_GC.tGenPrctTrip.GoodQual;
	IN_GC.tGen_LO_CoolingSys_Fail.Di	:=	IN_GC.tGen_LO_CoolingSys_Fail.Di 	OR NOT IN_GC.tGen_LO_CoolingSys_Fail.GoodQual;
	IN_GC.tGenCtr_CktBkr_Trip.Di		:=	IN_GC.tGenCtr_CktBkr_Trip.Di		OR NOT IN_GC.tGenCtr_CktBkr_Trip.GoodQual;
	IN_GC.tGenIF_CB_On.Di				:=	IN_GC.tGenIF_CB_On.Di				OR NOT IN_GC.tGenIF_CB_On.GoodQual;
	IN_GC.tGenHeat_CB_On.Di				:=	IN_GC.tGenHeat_CB_On.Di				OR NOT IN_GC.tGenHeat_CB_On.GoodQual;

	IN_GC.tLev_OilSkid_Sump_Hi.Di		:=	IN_GC.tLev_OilSkid_Sump_Hi.Di		OR NOT IN_GC.tLev_OilSkid_Sump_Hi.GoodQual;
	IN_GC.tDPr_OilSkid_FiltLP_Hi.Di		:=	IN_GC.tDPr_OilSkid_FiltLP_Hi.Di		OR NOT IN_GC.tDPr_OilSkid_FiltLP_Hi.GoodQual;
	IN_GC.tDPr_OilSkid_FiltHP_DE_Hi.Di	:=	IN_GC.tDPr_OilSkid_FiltHP_DE_Hi.Di	OR NOT IN_GC.tDPr_OilSkid_FiltHP_DE_Hi.GoodQual;
	IN_GC.tDPr_OilSkid_FiltHP_NDE_Hi.Di	:=	IN_GC.tDPr_OilSkid_FiltHP_NDE_Hi.Di	OR NOT IN_GC.tDPr_OilSkid_FiltHP_NDE_Hi.GoodQual;
	IN_GC.tOilSkid_PumpLP_CBOk.Di		:=	IN_GC.tOilSkid_PumpLP_CBOk.Di		OR NOT IN_GC.tOilSkid_PumpLP_CBOk.GoodQual;
	IN_GC.tOilSkid_PumpHP_CBOk.Di		:=	IN_GC.tOilSkid_PumpHP_CBOk.Di		OR NOT IN_GC.tOilSkid_PumpHP_CBOk.GoodQual;
	IN_GC.tOilSkid_PumpHP_CBOk_UPS.Di	:=	IN_GC.tOilSkid_PumpHP_CBOk_UPS.Di	OR NOT IN_GC.tOilSkid_PumpHP_CBOk_UPS.GoodQual;
	IN_GC.tOilSkid_Fan_CBOk.Di			:=	IN_GC.tOilSkid_Fan_CBOk.Di			OR NOT IN_GC.tOilSkid_Fan_CBOk.GoodQual;
	IN_GC.tOilSkid_Heater_CBOk.Di		:=	IN_GC.tOilSkid_Heater_CBOk.Di		OR NOT IN_GC.tOilSkid_Heater_CBOk.GoodQual;
	IN_GC.tOilSkid_MCB.Di				:=	IN_GC.tOilSkid_MCB.Di				OR NOT IN_GC.tOilSkid_MCB.GoodQual;
	IN_GC.tOilSkid_AuxV_Ok.Di			:=	IN_GC.tOilSkid_AuxV_Ok.Di			OR NOT IN_GC.tOilSkid_AuxV_Ok.GoodQual;
	IN_GC.tOilSkid_AuxV_Ok_UPS.Di		:=	IN_GC.tOilSkid_AuxV_Ok_UPS.Di		OR NOT IN_GC.tOilSkid_AuxV_Ok_UPS.GoodQual;
	IN_GC.tOilSkid_PumpC_CBOk.Di		:=	IN_GC.tOilSkid_PumpC_CBOk.Di		OR NOT IN_GC.tOilSkid_PumpC_CBOk.GoodQual;

	IN_GC.tP_GenRev_Ext.Di				:=	IN_GC.tP_GenRev_Ext.Di				OR	NOT IN_GC.tP_GenRev_Ext.GoodQual;
	IN_GC.tGenLossExc_Ext.Di			:=	IN_GC.tGenLossExc_Ext.Di			OR	NOT IN_GC.tGenLossExc_Ext.GoodQual;
	IN_GC.tU_GenAsy_Ext.Di				:=	IN_GC.tU_GenAsy_Ext.Di				OR	NOT IN_GC.tU_GenAsy_Ext.GoodQual;
	IN_GC.tI_GenAsy_Ext.Di				:=	IN_GC.tI_GenAsy_Ext.Di				OR	NOT IN_GC.tI_GenAsy_Ext.GoodQual;
	IN_GC.tGenOverExc.Di				:=	IN_GC.tGenOverExc.Di				OR	NOT IN_GC.tGenOverExc.GoodQual;
	IN_GC.tGenRotorEarthFault.Di		:=	IN_GC.tGenRotorEarthFault.Di		OR	NOT IN_GC.tGenRotorEarthFault.GoodQual;
	IN_GC.tQ_GenUnderVoltProt.Di		:=	IN_GC.tQ_GenUnderVoltProt.Di		OR	NOT IN_GC.tQ_GenUnderVoltProt.GoodQual;
	IN_GC.tGndFaultW.Di					:=	IN_GC.tGndFaultW.Di					OR	NOT IN_GC.tGndFaultW.GoodQual;
	IN_GC.tGenBearGreasSys2DE.Di		:=	IN_GC.tGenBearGreasSys2DE.Di		OR	NOT IN_GC.tGenBearGreasSys2DE.GoodQual;
	IN_GC.tGenBearGreasSys2NDE.Di		:=	IN_GC.tGenBearGreasSys2NDE.Di		OR	NOT IN_GC.tGenBearGreasSys2NDE.GoodQual;

END_PROGRAM
```

### Program Logical/Generator/general_GC (IEC, version 4.13.0) - general

#### general_GCCyclic.st
```iecst
(*******************************************************************************
general		general functions

This code is confidential AND proprietary to the INNIO Company.
It may NOT be used in any form, or reproduced in any manner,
without the express written permission of the INNIO Company.
Copyright, INNIO Company, 2022

Customized modifications: -
------------------------

History:
-------
V4.00.0	21.01.2015	lettenb.	new
V4.00.1	28.01.2015				release gen ctr included from pb8
V4.04.0	31.10.2016				tLeroySomer_AuxContactor.Do: Para.bU_adj_gcb_ext_hilo_a OR NOT Para.bU_adj_mcb_ext_hilo_a added
								(aufschaltung 110V referenzspg. verhindern bei verstellung mit AO/wasserer rosenheim)
V4.05.0	31.10.2017				parameter check for diagnosis added
V4.11.0	26.01.2022	lettenb.	IN_GC.bU_Set_NP_Rel added for change over to AVR voltage control
V4.13.0	20.11.2023	Farre,		added IN_GC.bBypassMCB_CosPhi and request power mode interfaces from CU needed for Microgrid (2023-168)

Instructions FOR use:
--------------------
Outstandings:
------------
*******************************************************************************)
PROGRAM _CYCLIC

	(* check para setup *)
	IN_GC.tPB2MM.bParaSetupOk;
	Para.iEng_Motortype;    (* MIN= 208   MAX= 920    *)
	Para.rN_EngStart_LimHi; (* MIN= 50.0  MAX= 2200.0 *)
	Para.iQ_GrC_CtrlFun;    (* MIN= 0     MAX= 8      *)
	Para.rF_Nom[1]; 		(* MIN= 49    MAX= 61     *)

	(* engine typ *)
	xEngType.Motortype := INT_TO_UINT(Para.iEng_Motortype);
	xEngType();				(* use: xEngType.Type2 as BOOL, ....*)

	(* engine operation mode *)
			bOMSS_Man  := FALSE;
			bOMSS_Aut  := FALSE;
			bOMSS_Test := FALSE;
			bOMSS_MAT  := FALSE;
			bOMSS_Scav := FALSE;
	CASE IN_GC.iIdx_OMSS OF
		1:	bOMSS_Man  := TRUE;
			bOMSS_MAT  := TRUE;
		2:	bOMSS_Aut  := TRUE;
			bOMSS_MAT  := TRUE;
		3:	bOMSS_Test := TRUE;
			bOMSS_MAT  := TRUE;
		4:	bOMSS_Scav := TRUE;
	END_CASE;

	(* PLC Running *)
	IN_GC.tPB2MM.bSys_Run;

	(* Operating mode *)
	xOpMode(in := IN_GC.iSt_OpMode);

	(*---------------------------------------------------------------------------*)
	(* start speed exceeded *)
	xGR_MAXR_DREHZ(In:= IN_GC.rN_EngAct, Gw:= Para.rN_EngStart_LimHi, Hy:= Para.rN_EngStart_HyHi);
	xTOF_M_DREHZ(IN:= xGR_MAXR_DREHZ.Q AND IN_GC.tPB2MM.bParaSetupOk, PT:= T#10s);
	M_DREHZ := xTOF_M_DREHZ.Q;

	(* ramp up speed *)
	xGR_MAXR_HDREHZ(In:= IN_GC.rN_EngAct, Gw:= Para.rN_EngStart_LimHiHi, Hy:= Para.rN_EngStart_HyHiHi);
	M_HDREHZ := xGR_MAXR_HDREHZ.Q AND IN_GC.tPB2MM.bParaSetupOk;

	(*---------------------------------------------------------------------------*)
	(* release AVR *)
	(* UNITROL: 0= U control/island mode, 1= Q control/mains parallel mode*)
	xGR_MAXR_AN_COS(In:= IN_GC.rP_Act_Norm_Filt, Gw:= Para.rGen_CosPhi_Ena, Hy:= Para.rGen_CosPhi_Ena_Hy);
	bGen_CosPhi_Ena := xGR_MAXR_AN_COS.Q AND IN_GC.tPB2MM.bParaSetupOk;

	OUT_GC.tPF_CosPCtr_Ena.Do :=   	bGen_CosPhi_Ena
							AND NOT IN_GC.bU_Set_NP_Rel
							AND 	IN_GC.tGCB_On.Di
							AND    (IN_GC.tMCB_On.Di OR (IN_GC.bReq_PowMod AND IN_GC.bOtherGenParallel) OR IN_GC.bBypassMCB_CosPhi);

	(* release voltage selection LS-generator *)
	OUT_GC.tLeroySomer_AuxContactor.Do :=  (IN_GC.bGen_SyD_Dem AND (NOT IN_GC.tGCB_On.Di           OR NOT IN_GC.tMCB_On.Di))
		 								OR (IN_GC.tGCB_DVM.Di  AND (NOT Para.bU_adj_gcb_ext_hilo_a OR NOT Para.bU_adj_mcb_ext_hilo_a))
		 								OR (IN_GC.tRel_U_Sel_LS_Gen.Di AND NOT Para.bSyActive);

	(* engine run + 30min *)
	xTON_Eng_Run_30m(IN	:= IN_GC.tEng_Run.Do, PT:= T#30m);
	bEng_Run_30m 		:= xTON_Eng_Run_30m.Q;						(* engine operation for 30 minutes *)

	(* Check if actual engine speed is zero *)
	bN_EngAct_IsZero	:= ((IN_GC.rN_EngAct > -0.01) AND (IN_GC.rN_EngAct < 0.01));

END_PROGRAM
```

#### general_GC.var
```iecst
VAR
	xGR_MAXR_AN_COS : GR_MAXR;
	xGR_MAXR_DREHZ : GR_MAXR;
	xGR_MAXR_HDREHZ : GR_MAXR;
	xTOF_M_DREHZ : TOF;
	xTON_Eng_Run_30m : TON := (0); (*FuB*)
END_VAR
```

### Program Logical/Generator/ereg (IEC, version 4.10.0) - excitation

#### eregCyclicst.st
```iecst
(********************************************************************
ereg	 			 generator excitation voltage

This code is confidential and proprietary to the INNIO Company.
It may not be used in any form, or reproduced in any manner,
without written permission of the INNIO Company.
Copyright, INNIO Company, 2019

Customized modifications: -
------------------------

History:
-------

V0.1  	27.10.98/Pa	  			Created
      	24.11.98/Pa	  			Proofread
V170  	15.04.02/LH	  			Delay in excitation voltage minimum => 10sec
V180  	06.03.03/LH	  			VISU- Limit values only after recipe is on controller
      	18.03.03/LH	  			Read analog input -> pb17
V190  	19.04.04/LH	  			Limit value excitation voltage maximum
V350  	25.02.13/HG,IG  		Modular software - new "english" names, moved filtering & scaling to HAL
		06.06.2016	lettenb.	M_DREHZ added, set value to zero if engine stand still acc.XT3, bugfix
V4.10.0	14.12.2020	lettenb.	TON,TOF reset added to avoid time overrun, cleanup

Instructions for use: -
--------------------

Outstandings:
------------

*******************************************************************************)

PROGRAM _CYCLIC

	IF Para.bU_Gen_Exc_Ena AND M_DREHZ THEN
		(* Generator excitation activated *)

		(* Set point excitation voltage minimum *)
		xGRMinFA_AN_ERGW1.In := IN_GC.tU_Gen_Exc.Ai;
		xGRMinFA_AN_ERGW1.Gw := Para.rU_Gen_ExcLo;
		xGRMinFA_AN_ERGW1.Hy := Para.rU_Gen_ExcHyLo;
		xGRMinFA_AN_ERGW1();
		xTON_FA_T_ERGW1.IN   := xGRMinFA_AN_ERGW1.Q AND IN_GC.tPB2MM.bParaSetupOk;
		xTON_FA_T_ERGW1.PT   := T#10s;
		xTON_FA_T_ERGW1();
		bU_Gen_Exc_Min       := xTON_FA_T_ERGW1.Q;

		(* Set point excitation voltage maximum *)
		xGRMaxFA_AN_ERGW2.In := IN_GC.tU_Gen_Exc.Ai;
		xGRMaxFA_AN_ERGW2.Gw := Para.rU_Gen_ExcHi;
		xGRMaxFA_AN_ERGW2.Hy := Para.rU_Gen_ExcHyHi;
		xGRMaxFA_AN_ERGW2();
		xTON_FA_T_ERGW2.IN   := xGRMaxFA_AN_ERGW2.Q AND IN_GC.tPB2MM.bParaSetupOk;
		xTON_FA_T_ERGW2.PT   := T#30s;
		xTON_FA_T_ERGW2();
		bU_Gen_Exc_Max       := xTON_FA_T_ERGW2.Q;

		OUT_GC.rU_Gen_Exc    := IN_GC.tU_Gen_Exc.Ai;

	ELSE
		xTON_FA_T_ERGW1(IN:= FALSE, PT:= T#0s);
		xTON_FA_T_ERGW2(IN:= FALSE, PT:= T#0s);

		bU_Gen_Exc_Min     := FALSE;
		bU_Gen_Exc_Max     := FALSE;
		OUT_GC.rU_Gen_Exc  := 0.0;

	END_IF;

END_PROGRAM
```

#### ereg.var
```iecst
VAR
	xGRMaxFA_AN_ERGW2 : GR_MAXR;
	xGRMinFA_AN_ERGW1 : GR_MINR;
	xTON_FA_T_ERGW2 : TON;
	xTON_FA_T_ERGW1 : TON;
END_VAR
```

### Program Logical/Generator/gwt (IEC, version 4.07.0) - gen.winding temperature

#### gwtCyclicst.st
```iecst
(********************************************************************
gwt	 	Generator: winding temp.monitoring/bearing temp.monitoring

This code is confidential and proprietary to the INNIO Company.
It may not be used in any form, or reproduced in any manner,
without written permission of the INNIO Company.
Copyright, INNIO Company, 2019

Customized modifications: -
------------------------
History:
-------

Winding temperature AND Bearing temperature
_______________________________________________________________________________________
VER	Datum/Name	Änderung
V0.1	21.10.1998	Pa			Created
 	    26.11.1998	Pa			Proofread
V180	06.03.2003	LH			VISU - Limit values active only when Recipes are on controller
 	    18.03.2003	LH			Reading the analog inputs -> pb17
V210	24.11.2004	LH			Bit to display winding temperature with measurement point 1
V2100b	15.09.2006	LH			Bit to display winding temperature with 1 measurement switched off,
				    			if 1 measurement point is with PT100 switched off.
V220	20.04.2007	LH			Bit to display Winding temperature mit 1 measurement point -> "settings"
V2201	23.07.2007	LH			Measurement signal winding 1 - phase : Lower limit changed from -20°C to --> -50°C
		23.07.2007	LH			Measurement signal winding 3 - phase : Lower limit changed from -20°C to --> -50°C
														   Upper limit changed from 200°C to --> 230°C
		23.07.2007	LH			Measurement signal bearing temperature : Lower limit changed from -20°C to --> -50°C
V4.00.1	28.01.2014	lettenb.	code cleanup
V4.05.0	14.12.2017	lettenb.	write parameter removed(code guide line)cleanup
V4.07.0	24.06.2019	lettenb.	xGR_MAXR_FA_AN_GW_TW added for SP Winding temperature warning, bugfix

Instructions for use: -
--------------------
Outstandings:
------------
*******************************************************************************)

PROGRAM _CYCLIC

	IF NOT Para.bT_Gen_Wind_Ena THEN
		// 3 Phase monitoring NOT turned on, reset unused interfaces

		bT_Gen_Wind_L1_Max := FALSE;
		bT_Gen_Wind_L2_Max := FALSE;
		bT_Gen_Wind_L3_Max := FALSE;

		bT_Gen_Wind_L1_Lim := FALSE;
		bT_Gen_Wind_L2_Lim := FALSE;
		bT_Gen_Wind_L3_Lim := FALSE;

		(* SP Winding temperature trip *)
		xGR_MAXR_FA_AN_GW_TA(In:= IN_GC.tT_Gen_Wind.Ai, Gw:= Para.rT_Gen_Wind_Max, Hy:= Para.rT_Gen_Wind_Max_Hy2);
		xTON_FA_AN_GWTA(IN:= xGR_MAXR_FA_AN_GW_TA.Q AND IN_GC.tPB2MM.bParaSetupOk, PT:= T#2s);
		bT_Gen_Wind_Max := xTON_FA_AN_GWTA.Q;

		(* SP Winding temperature warning *)
		xGR_MAXR_FA_AN_GW_TW(In:= IN_GC.tT_Gen_Wind.Ai, Gw:= Para.rT_Gen_Wind_Lim, Hy:= Para.rT_Gen_Wind_Lim_Hy);
		xTON_FA_AN_GWTW(IN:= xGR_MAXR_FA_AN_GW_TW.Q AND IN_GC.tPB2MM.bParaSetupOk, PT:= T#2s);
		bT_Gen_Wind_Lim := xTON_FA_AN_GWTW.Q;

	ELSE
		// 1-Phase Monitoring inactive
		// 3-Phase monitoring   active

		bT_Gen_Wind_Max := FALSE;
		bT_Gen_Wind_Lim := FALSE;

		(* SP Winding 1 temperature warning *)
		xGR_MAXR_FA_GWW1(In:= IN_GC.tT_Gen_Wind_Act_L1.Ai, Gw:= Para.rT_Gen_Wind_Lim_L1, Hy:= Para.rT_Gen_Wind_Lim_Hy2);
		xTON_FA_AN_GWW1(IN:= xGR_MAXR_FA_GWW1.Q AND IN_GC.tPB2MM.bParaSetupOk, PT:= T#2s);
		bT_Gen_Wind_L1_Lim := xTON_FA_AN_GWW1.Q;

		(* SP Winding 2 temperature warning *)
		xGR_MAXR_FA_GWW2(In:= IN_GC.tT_Gen_Wind_Act_L2.Ai, Gw:= Para.rT_Gen_Wind_Lim_L2, Hy:= Para.rT_Gen_Wind_Lim_Hy2);
		xTON_FA_AN_GWW2(IN:= xGR_MAXR_FA_GWW2.Q AND IN_GC.tPB2MM.bParaSetupOk, PT:= T#2s);
		bT_Gen_Wind_L2_Lim := xTON_FA_AN_GWW2.Q;

		(* SP Winding 3 temperature warning *)
		xGR_MAXR_FA_GWW3(In:= IN_GC.tT_Gen_Wind_Act_L3.Ai, Gw:= Para.rT_Gen_Wind_Lim_L3, Hy:= Para.rT_Gen_Wind_Lim_Hy2);
		xTON_FA_AN_GWW3(IN:= xGR_MAXR_FA_GWW3.Q AND IN_GC.tPB2MM.bParaSetupOk, PT:= T#3s);
		bT_Gen_Wind_L3_Lim := xTON_FA_AN_GWW3.Q;

		(* SP Winding 1 temperature trip *)
		xGR_MAXR_FA_GWA1(In:= IN_GC.tT_Gen_Wind_Act_L1.Ai, Gw:= Para.rT_Gen_Wind_Max_L1, Hy:= Para.rT_Gen_Wind_Max_Hy);
		xTON_FA_T_AN_GWA1(IN:= xGR_MAXR_FA_GWA1.Q AND IN_GC.tPB2MM.bParaSetupOk, PT:= T#2s);
		bT_Gen_Wind_L1_Max := xTON_FA_T_AN_GWA1.Q;

		(* SP Winding 2 temperature trip *)
		xGR_MAXR_FA_GWA2(In:= IN_GC.tT_Gen_Wind_Act_L2.Ai, Gw:= Para.rT_Gen_Wind_Max_L2, Hy:= Para.rT_Gen_Wind_Max_Hy);
		xTON_FA_T_AN_GWA2(IN:= xGR_MAXR_FA_GWA2.Q AND IN_GC.tPB2MM.bParaSetupOk, PT:= T#2s);
		bT_Gen_Wind_L2_Max := xTON_FA_T_AN_GWA2.Q;

		(* SP Winding 3 temperature trip *)
		xGR_MAXR_FA_GWA3(In:= IN_GC.tT_Gen_Wind_Act_L3.Ai, Gw:= Para.rT_Gen_Wind_Max_L3, Hy:= Para.rT_Gen_Wind_Max_Hy);
		xTON_FA_T_AN_GWA3(IN:= xGR_MAXR_FA_GWA3.Q AND IN_GC.tPB2MM.bParaSetupOk, PT:= T#3s);
		bT_Gen_Wind_L3_Max := xTON_FA_T_AN_GWA3.Q;

	END_IF;

(*
   There can be total of two bearing temperature monitors.
   Based on the Para.bT_Gen_Bear_A_Ena and Para.bT_Gen_Bear_B_Ena parameters it is possible to monitor
	 1. One of the bearing temperature
 	 2. Both bearing temperatures
	 3. None of the bearing temperatures (if not required eg. low KW engines)
*)

	(* Bearing1 temperature monitoring *)
	IF NOT Para.bT_Gen_Bear_A_Ena THEN 	(* Bearing temperature monitoring inactive *)
		bT_Gen_Bear_A_Max := FALSE;
		bT_Gen_Bear_A_Lim := FALSE;
	ELSE								(* Bearing temperature monitoring active *)
		(* Bearing 1 Temperature maximum Warning *)
		xGR_MAXR_FA_AN_LAGW1(In:= IN_GC.tT_Gen_Bear_A_Act.Ai, Gw:= Para.rT_Gen_Bear_Lim_A, Hy:= Para.rT_Gen_Bear_Max_Hy_A);
		xTON_FA_T_AN_LAGW1(IN:= xGR_MAXR_FA_AN_LAGW1.Q AND IN_GC.tPB2MM.bParaSetupOk, PT:= T#2s);
		bT_Gen_Bear_A_Lim := xTON_FA_T_AN_LAGW1.Q;

		(* Bearing 1 Temperature maximum Trip*)
		xGR_MAXR_FA_AN_LAGA1(In:= IN_GC.tT_Gen_Bear_A_Act.Ai, Gw:= Para.rT_Gen_Bear_Max_A, Hy:= Para.rT_Gen_Bear_Max_Hy_A);
		xTON_FA_T_AN_LAGA1(IN:= xGR_MAXR_FA_AN_LAGA1.Q AND IN_GC.tPB2MM.bParaSetupOk, PT:= T#2s);
		bT_Gen_Bear_A_Max := xTON_FA_T_AN_LAGA1.Q;
	END_IF;

	(* Bearing2 temperature monitoring *)
	IF NOT Para.bT_Gen_Bear_B_Ena THEN	(* Bearing temperature monitoring inactive	*)
		bT_Gen_Bear_B_Max := FALSE;
		bT_Gen_Bear_B_Lim := FALSE;
	ELSE								(* Bearing temperature monitoring active *)
		(* SP Bearing 2 Temperature maximum Warning *)
		xGR_MAXR_FA_AN_LAGW2(In:= IN_GC.tT_Gen_Bear_B_Act.Ai, Gw:= Para.rT_Gen_Bear_Lim_B, Hy:= Para.rT_Gen_Bear_Max_Hy_B);
		xTON_FA_T_AN_LAGW2(IN:= xGR_MAXR_FA_AN_LAGW2.Q AND IN_GC.tPB2MM.bParaSetupOk, PT:= T#2s);
		bT_Gen_Bear_B_Lim := xTON_FA_T_AN_LAGW2.Q;

		(* SP Bearing 2 Temperature maximum Trip*)
		xGR_MAXR_FA_AN_LAGA2(In:= IN_GC.tT_Gen_Bear_B_Act.Ai, Gw:= Para.rT_Gen_Bear_Max_B, Hy:= Para.rT_Gen_Bear_Max_Hy_B);
		xTON_FA_T_AN_LAGA2(IN:= xGR_MAXR_FA_AN_LAGA2.Q AND IN_GC.tPB2MM.bParaSetupOk, PT:= T#2s);
		bT_Gen_Bear_B_Max := xTON_FA_T_AN_LAGA2.Q;
	END_IF;

END_PROGRAM
```

#### gwtInitst.st
```iecst
(********************************************************************
gwt	 			 Initialization

This code is confidential and proprietary to the INNIO Company.
It may not be used in any form, or reproduced in any manner,
without written permission of the INNIO Company.
Copyright, INNIO Company, 2019

Customized modifications: -
------------------------

History:
-------

Instructions for use: -
--------------------

Outstandings:
------------

*******************************************************************************)

PROGRAM _INIT

END_PROGRAM
```
